P[382]{
   GP1:
	UF : 0, UT : 1,		CONFIG : 'N U T, 0, 0, 0',
	X =	1901.936766	mm,	Y =	727.255833	mm,	Z =	782.023540	mm,
	W =	-151.714705	deg,	P =	-51.403130	deg,	R =	86.436087	deg
};
P[383]{
   GP1:
	UF : 0, UT : 1,		CONFIG : 'N U T, 0, 0, 0',
	X =	1885.131021	mm,	Y =	717.571438	mm,	Z =	785.030103	mm,
	W =	-147.037443	deg,	P =	-51.128385	deg,	R =	85.635377	deg
};
P[384]{
   GP1:
	UF : 0, UT : 1,		CONFIG : 'N U T, 0, 0, 0',
	X =	1869.049725	mm,	Y =	707.056034	mm,	Z =	788.968292	mm,
	W =	-142.293668	deg,	P =	-50.578645	deg,	R =	84.961258	deg
};
P[385]{
   GP1:
	UF : 0, UT : 1,		CONFIG : 'N U T, 0, 0, 0',
	X =	1853.457899	mm,	Y =	695.952416	mm,	Z =	793.610294	mm,
	W =	-139.371378	deg,	P =	-49.801635	deg,	R =	84.946616	deg
};
P[386]{
   GP1:
	UF : 0, UT : 1,		CONFIG : 'N U T, 0, 0, 0',
	X =	1838.594903	mm,	Y =	684.232405	mm,	Z =	798.951702	mm,
	W =	-135.684529	deg,	P =	-49.179213	deg,	R =	84.598217	deg
};
P[387]{
   GP1:
	UF : 0, UT : 1,		CONFIG : 'N U T, 0, 0, 0',
	X =	1824.247050	mm,	Y =	672.047896	mm,	Z =	804.854588	mm,
	W =	-133.003710	deg,	P =	-48.647484	deg,	R =	84.428097	deg
};
P[388]{
   GP1:
	UF : 0, UT : 1,		CONFIG : 'N U T, 0, 0, 0',
	X =	1810.719043	mm,	Y =	659.440410	mm,	Z =	811.371247	mm,
	W =	-129.945774	deg,	P =	-47.843357	deg,	R =	84.483658	deg
};
P[389]{
   GP1:
	UF : 0, UT : 1,		CONFIG : 'N U T, 0, 0, 0',
	X =	1804.034364	mm,	Y =	652.928161	mm,	Z =	814.783583	mm,
	W =	-128.085999	deg,	P =	-47.790016	deg,	R =	83.961023	deg
};
P[390]{
   GP1:
	UF : 0, UT : 1,		CONFIG : 'N U T, 0, 0, 0',
	X =	1805.489552	mm,	Y =	648.057612	mm,	Z =	805.993139	mm,
	W =	-118.280441	deg,	P =	-25.249973	deg,	R =	66.929569	deg
};
P[391]{
   GP1:
	UF : 0, UT : 1,		CONFIG : 'N U T, 0, 0, 0',
	X =	1812.203439	mm,	Y =	654.534929	mm,	Z =	802.566706	mm,
	W =	-118.280441	deg,	P =	-25.249973	deg,	R =	66.929569	deg
};
P[392]{
   GP1:
	UF : 0, UT : 1,		CONFIG : 'N U T, 0, 0, 0',
	X =	1825.953302	mm,	Y =	667.117557	mm,	Z =	796.150605	mm,
	W =	-119.553021	deg,	P =	-25.967899	deg,	R =	66.217655	deg
};
P[393]{
   GP1:
	UF : 0, UT : 1,		CONFIG : 'N U T, 0, 0, 0',
	X =	1840.283003	mm,	Y =	679.245035	mm,	Z =	790.296569	mm,
	W =	-121.343606	deg,	P =	-27.066084	deg,	R =	65.126643	deg
};
P[394]{
   GP1:
	UF : 0, UT : 1,		CONFIG : 'N U T, 0, 0, 0',
	X =	1855.178855	mm,	Y =	690.957511	mm,	Z =	785.030157	mm,
	W =	-123.834308	deg,	P =	-27.839914	deg,	R =	64.621906	deg
};
P[395]{
   GP1:
	UF : 0, UT : 1,		CONFIG : 'N U T, 0, 0, 0',
	X =	1870.722402	mm,	Y =	702.006487	mm,	Z =	780.427067	mm,
	W =	-125.757358	deg,	P =	-29.362690	deg,	R =	63.090015	deg
};
P[396]{
   GP1:
	UF : 0, UT : 1,		CONFIG : 'N U T, 0, 0, 0',
	X =	1886.912120	mm,	Y =	712.361926	mm,	Z =	776.544794	mm,
	W =	-127.137960	deg,	P =	-31.279411	deg,	R =	61.084884	deg
};
P[397]{
   GP1:
	UF : 0, UT : 1,		CONFIG : 'N U T, 0, 0, 0',
	X =	1903.741024	mm,	Y =	721.914625	mm,	Z =	773.719192	mm,
	W =	-130.946538	deg,	P =	-32.608966	deg,	R =	60.232135	deg
};
P[398]{
   GP1:
	UF : 0, UT : 1,		CONFIG : 'N U T, 0, 0, 0',
	X =	1921.157911	mm,	Y =	730.631468	mm,	Z =	771.649972	mm,
	W =	-133.177286	deg,	P =	-34.370572	deg,	R =	58.698336	deg
};
P[399]{
   GP1:
	UF : 0, UT : 1,		CONFIG : 'N U T, 0, 0, 0',
	X =	1939.106460	mm,	Y =	738.185459	mm,	Z =	770.748033	mm,
	W =	-136.382473	deg,	P =	-36.661003	deg,	R =	56.846048	deg
};
P[400]{
   GP1:
	UF : 0, UT : 1,		CONFIG : 'N U T, 0, 0, 0',
	X =	1957.509282	mm,	Y =	744.705160	mm,	Z =	770.921949	mm,
	W =	-140.117439	deg,	P =	-38.294588	deg,	R =	55.735219	deg
};
P[401]{
   GP1:
	UF : 0, UT : 1,		CONFIG : 'N U T, 0, 0, 0',
	X =	1976.233128	mm,	Y =	749.875221	mm,	Z =	772.261698	mm,
	W =	-143.501798	deg,	P =	-40.756036	deg,	R =	53.888603	deg
};
P[402]{
   GP1:
	UF : 0, UT : 1,		CONFIG : 'N U T, 0, 0, 0',
	X =	1995.151040	mm,	Y =	753.608286	mm,	Z =	774.825499	mm,
	W =	-146.537598	deg,	P =	-43.694495	deg,	R =	51.728917	deg
};
P[403]{
   GP1:
	UF : 0, UT : 1,		CONFIG : 'N U T, 0, 0, 0',
	X =	2014.131662	mm,	Y =	756.050102	mm,	Z =	778.522436	mm,
	W =	-149.631146	deg,	P =	-46.183910	deg,	R =	50.037999	deg
};
P[404]{
   GP1:
	UF : 0, UT : 1,		CONFIG : 'N U T, 0, 0, 0',
	X =	2032.817354	mm,	Y =	756.903352	mm,	Z =	783.674625	mm,
	W =	-155.609996	deg,	P =	-47.899495	deg,	R =	49.040964	deg
};
P[405]{
   GP1:
	UF : 0, UT : 1,		CONFIG : 'N U T, 0, 0, 0',
	X =	2051.302092	mm,	Y =	756.193182	mm,	Z =	789.739862	mm,
	W =	-157.425664	deg,	P =	-51.603070	deg,	R =	46.654443	deg
};
P[406]{
   GP1:
	UF : 0, UT : 1,		CONFIG : 'N U T, 0, 0, 0',
	X =	2069.427420	mm,	Y =	754.378399	mm,	Z =	796.789881	mm,
	W =	-160.571018	deg,	P =	-53.566344	deg,	R =	45.491306	deg
};
P[407]{
   GP1:
	UF : 0, UT : 1,		CONFIG : 'N U T, 0, 0, 0',
	X =	2086.942757	mm,	Y =	751.238839	mm,	Z =	804.750806	mm,
	W =	-163.790463	deg,	P =	-56.037649	deg,	R =	44.063831	deg
};
P[408]{
   GP1:
	UF : 0, UT : 1,		CONFIG : 'N U T, 0, 0, 0',
	X =	2103.734538	mm,	Y =	746.847799	mm,	Z =	813.628016	mm,
	W =	-167.805714	deg,	P =	-57.866850	deg,	R =	42.962546	deg
};
P[409]{
   GP1:
	UF : 0, UT : 1,		CONFIG : 'N U T, 0, 0, 0',
	X =	2120.121828	mm,	Y =	741.533562	mm,	Z =	823.012356	mm,
	W =	-169.515653	deg,	P =	-59.824191	deg,	R =	41.934243	deg
};
P[410]{
   GP1:
	UF : 0, UT : 1,		CONFIG : 'N U T, 0, 0, 0',
	X =	2135.809632	mm,	Y =	735.266252	mm,	Z =	832.922306	mm,
	W =	-170.897609	deg,	P =	-62.624007	deg,	R =	40.637323	deg
};
P[411]{
   GP1:
	UF : 0, UT : 1,		CONFIG : 'N U T, 0, 0, 0',
	X =	2150.697320	mm,	Y =	728.173791	mm,	Z =	843.480209	mm,
	W =	-174.130853	deg,	P =	-63.898821	deg,	R =	39.881575	deg
};
P[412]{
   GP1:
	UF : 0, UT : 1,		CONFIG : 'N U T, 0, 0, 0',
	X =	2165.138622	mm,	Y =	720.374642	mm,	Z =	854.327618	mm,
	W =	-175.204728	deg,	P =	-65.758106	deg,	R =	39.148980	deg
};
P[413]{
   GP1:
	UF : 0, UT : 1,		CONFIG : 'N U T, 0, 0, 0',
	X =	2178.740148	mm,	Y =	711.855194	mm,	Z =	865.589791	mm,
	W =	-177.331694	deg,	P =	-67.680964	deg,	R =	38.363196	deg
};
P[414]{
   GP1:
	UF : 0, UT : 1,		CONFIG : 'N U T, 0, 0, 0',
	X =	2191.774572	mm,	Y =	702.742815	mm,	Z =	877.172249	mm,
	W =	-178.961511	deg,	P =	-69.127925	deg,	R =	37.827748	deg
};
P[415]{
   GP1:
	UF : 0, UT : 1,		CONFIG : 'N U T, 0, 0, 0',
	X =	2186.634600	mm,	Y =	701.073329	mm,	Z =	863.753783	mm,
	W =	133.613067	deg,	P =	-56.139818	deg,	R =	90.707230	deg
};
P[416]{
   GP1:
	UF : 0, UT : 1,		CONFIG : 'N U T, 0, 0, 0',
	X =	2173.210709	mm,	Y =	710.002963	mm,	Z =	852.229285	mm,
	W =	133.613067	deg,	P =	-56.139818	deg,	R =	90.707230	deg
};
P[417]{
   GP1:
	UF : 0, UT : 1,		CONFIG : 'N U T, 0, 0, 0',
	X =	2159.155826	mm,	Y =	718.028851	mm,	Z =	841.201692	mm,
	W =	136.846302	deg,	P =	-55.948190	deg,	R =	91.020186	deg
};
P[418]{
   GP1:
	UF : 0, UT : 1,		CONFIG : 'N U T, 0, 0, 0',
	X =	2144.534743	mm,	Y =	725.561610	mm,	Z =	830.433379	mm,
	W =	139.007318	deg,	P =	-55.906508	deg,	R =	91.308868	deg
};
P[419]{
   GP1:
	UF : 0, UT : 1,		CONFIG : 'N U T, 0, 0, 0',
	X =	2129.236263	mm,	Y =	732.215606	mm,	Z =	820.204356	mm,
	W =	142.641369	deg,	P =	-55.588173	deg,	R =	91.285535	deg
};
P[420]{
   GP1:
	UF : 0, UT : 1,		CONFIG : 'N U T, 0, 0, 0',
	X =	2113.285254	mm,	Y =	738.059573	mm,	Z =	810.455841	mm,
	W =	146.014779	deg,	P =	-55.372652	deg,	R =	91.325542	deg
};
P[421]{
   GP1:
	UF : 0, UT : 1,		CONFIG : 'N U T, 0, 0, 0',
	X =	2096.698526	mm,	Y =	742.938558	mm,	Z =	801.332479	mm,
	W =	149.978045	deg,	P =	-55.027116	deg,	R =	91.206586	deg
};
P[422]{
   GP1:
	UF : 0, UT : 1,		CONFIG : 'N U T, 0, 0, 0',
	X =	2079.499669	mm,	Y =	746.762081	mm,	Z =	792.911791	mm,
	W =	154.264576	deg,	P =	-54.635969	deg,	R =	91.033179	deg
};
P[423]{
   GP1:
	UF : 0, UT : 1,		CONFIG : 'N U T, 0, 0, 0',
	X =	2061.718554	mm,	Y =	749.294435	mm,	Z =	785.384968	mm,
	W =	159.358992	deg,	P =	-54.241219	deg,	R =	90.849508	deg
};
P[424]{
   GP1:
	UF : 0, UT : 1,		CONFIG : 'N U T, 0, 0, 0',
	X =	2043.468705	mm,	Y =	750.695013	mm,	Z =	778.604240	mm,
	W =	163.651309	deg,	P =	-54.643114	deg,	R =	91.026912	deg
};
P[425]{
   GP1:
	UF : 0, UT : 1,		CONFIG : 'N U T, 0, 0, 0',
	X =	2024.862362	mm,	Y =	750.526321	mm,	Z =	773.152849	mm,
	W =	170.177142	deg,	P =	-53.461414	deg,	R =	90.339652	deg
};
P[426]{
   GP1:
	UF : 0, UT : 1,		CONFIG : 'N U T, 0, 0, 0',
	X =	2005.984397	mm,	Y =	748.955899	mm,	Z =	768.770108	mm,
	W =	175.722594	deg,	P =	-52.709076	deg,	R =	89.957307	deg
};
P[427]{
   GP1:
	UF : 0, UT : 1,		CONFIG : 'N U T, 0, 0, 0',
	X =	1987.047314	mm,	Y =	746.010534	mm,	Z =	765.364078	mm,
	W =	-178.653351	deg,	P =	-53.676796	deg,	R =	89.597607	deg
};
P[428]{
   GP1:
	UF : 0, UT : 1,		CONFIG : 'N U T, 0, 0, 0',
	X =	1968.269258	mm,	Y =	741.589641	mm,	Z =	763.449879	mm,
	W =	-172.301934	deg,	P =	-52.215645	deg,	R =	89.108243	deg
};
P[429]{
   GP1:
	UF : 0, UT : 1,		CONFIG : 'N U T, 0, 0, 0',
	X =	1949.683228	mm,	Y =	735.867392	mm,	Z =	762.574025	mm,
	W =	-166.727696	deg,	P =	-52.147337	deg,	R =	88.499624	deg
};
P[430]{
   GP1:
	UF : 0, UT : 1,		CONFIG : 'N U T, 0, 0, 0',
	X =	1931.537687	mm,	Y =	728.906759	mm,	Z =	762.984667	mm,
	W =	-161.402140	deg,	P =	-50.785190	deg,	R =	88.352660	deg
};
P[431]{
   GP1:
	UF : 0, UT : 1,		CONFIG : 'N U T, 0, 0, 0',
	X =	1913.894369	mm,	Y =	720.759021	mm,	Z =	764.365662	mm,
	W =	-155.472702	deg,	P =	-51.263880	deg,	R =	87.224493	deg
};
P[432]{
   GP1:
	UF : 0, UT : 1,		CONFIG : 'N U T, 0, 0, 0',
	X =	1896.775808	mm,	Y =	711.703886	mm,	Z =	766.784223	mm,
	W =	-150.833605	deg,	P =	-50.652086	deg,	R =	86.780879	deg
};
P[433]{
   GP1:
	UF : 0, UT : 1,		CONFIG : 'N U T, 0, 0, 0',
	X =	1880.295912	mm,	Y =	701.786455	mm,	Z =	770.150545	mm,
	W =	-146.630492	deg,	P =	-49.748494	deg,	R =	86.649965	deg
};
P[434]{
   GP1:
	UF : 0, UT : 1,		CONFIG : 'N U T, 0, 0, 0',
	X =	1864.365138	mm,	Y =	691.155671	mm,	Z =	774.234987	mm,
	W =	-142.794729	deg,	P =	-49.424405	deg,	R =	86.125445	deg
};
P[435]{
   GP1:
	UF : 0, UT : 1,		CONFIG : 'N U T, 0, 0, 0',
	X =	1849.113413	mm,	Y =	679.894582	mm,	Z =	779.109083	mm,
	W =	-139.403776	deg,	P =	-48.562422	deg,	R =	86.186590	deg
};
P[436]{
   GP1:
	UF : 0, UT : 1,		CONFIG : 'N U T, 0, 0, 0',
	X =	1834.491060	mm,	Y =	668.059164	mm,	Z =	784.620839	mm,
	W =	-136.088896	deg,	P =	-48.063889	deg,	R =	85.921463	deg
};
P[437]{
   GP1:
	UF : 0, UT : 1,		CONFIG : 'N U T, 0, 0, 0',
	X =	1820.513635	mm,	Y =	655.728175	mm,	Z =	790.732302	mm,
	W =	-132.837127	deg,	P =	-47.655336	deg,	R =	85.548407	deg
};
P[438]{
   GP1:
	UF : 0, UT : 1,		CONFIG : 'N U T, 0, 0, 0',
	X =	1807.025014	mm,	Y =	643.027015	mm,	Z =	797.323227	mm,
	W =	-130.462952	deg,	P =	-47.253573	deg,	R =	85.381539	deg
};
P[439]{
   GP1:
	UF : 0, UT : 1,		CONFIG : 'N U T, 0, 0, 0',
	X =	1808.632578	mm,	Y =	637.999708	mm,	Z =	788.721272	mm,
	W =	-119.968116	deg,	P =	-24.932390	deg,	R =	67.755263	deg
};
P[440]{
   GP1:
	UF : 0, UT : 1,		CONFIG : 'N U T, 0, 0, 0',
	X =	1815.310699	mm,	Y =	644.342823	mm,	Z =	785.396809	mm,
	W =	-119.968116	deg,	P =	-24.932390	deg,	R =	67.755263	deg
};
P[441]{
   GP1:
	UF : 0, UT : 1,		CONFIG : 'N U T, 0, 0, 0',
	X =	1828.937900	mm,	Y =	656.757079	mm,	Z =	779.075124	mm,
	W =	-120.933291	deg,	P =	-25.503310	deg,	R =	67.152954	deg
};
P[442]{
   GP1:
	UF : 0, UT : 1,		CONFIG : 'N U T, 0, 0, 0',
	X =	1843.195636	mm,	Y =	668.591056	mm,	Z =	773.448643	mm,
	W =	-123.046463	deg,	P =	-26.806027	deg,	R =	65.806724	deg
};
P[443]{
   GP1:
	UF : 0, UT : 1,		CONFIG : 'N U T, 0, 0, 0',
	X =	1858.023543	mm,	Y =	680.021234	mm,	Z =	768.338080	mm,
	W =	-124.862562	deg,	P =	-27.804666	deg,	R =	64.848593	deg
};
P[444]{
   GP1:
	UF : 0, UT : 1,		CONFIG : 'N U T, 0, 0, 0',
	X =	1873.459502	mm,	Y =	690.849611	mm,	Z =	763.968271	mm,
	W =	-127.624928	deg,	P =	-28.905108	deg,	R =	63.936758	deg
};
P[445]{
   GP1:
	UF : 0, UT : 1,		CONFIG : 'N U T, 0, 0, 0',
	X =	1889.485011	mm,	Y =	701.051034	mm,	Z =	760.200825	mm,
	W =	-129.215229	deg,	P =	-30.446290	deg,	R =	62.373977	deg
};
P[446]{
   GP1:
	UF : 0, UT : 1,		CONFIG : 'N U T, 0, 0, 0',
	X =	1906.116311	mm,	Y =	710.431489	mm,	Z =	757.393894	mm,
	W =	-132.248082	deg,	P =	-32.023439	deg,	R =	61.033740	deg
};
P[447]{
   GP1:
	UF : 0, UT : 1,		CONFIG : 'N U T, 0, 0, 0',
	X =	1923.335471	mm,	Y =	718.930100	mm,	Z =	755.412367	mm,
	W =	-134.227112	deg,	P =	-34.097959	deg,	R =	59.112079	deg
};
P[448]{
   GP1:
	UF : 0, UT : 1,		CONFIG : 'N U T, 0, 0, 0',
	X =	1941.074451	mm,	Y =	726.336330	mm,	Z =	754.576473	mm,
	W =	-137.427428	deg,	P =	-36.272612	deg,	R =	57.336758	deg
};
P[449]{
   GP1:
	UF : 0, UT : 1,		CONFIG : 'N U T, 0, 0, 0',
	X =	1959.258358	mm,	Y =	732.705571	mm,	Z =	754.756467	mm,
	W =	-140.534645	deg,	P =	-38.203158	deg,	R =	55.855613	deg
};
P[450]{
   GP1:
	UF : 0, UT : 1,		CONFIG : 'N U T, 0, 0, 0',
	X =	1977.709684	mm,	Y =	737.832473	mm,	Z =	756.240512	mm,
	W =	-145.990036	deg,	P =	-39.401021	deg,	R =	55.158578	deg
};
P[451]{
   GP1:
	UF : 0, UT : 1,		CONFIG : 'N U T, 0, 0, 0',
	X =	1996.381049	mm,	Y =	741.462266	mm,	Z =	758.804472	mm,
	W =	-148.889992	deg,	P =	-42.355562	deg,	R =	52.899958	deg
};
P[452]{
   GP1:
	UF : 0, UT : 1,		CONFIG : 'N U T, 0, 0, 0',
	X =	2015.092255	mm,	Y =	743.714069	mm,	Z =	762.512016	mm,
	W =	-151.386913	deg,	P =	-45.459649	deg,	R =	50.658130	deg
};
P[453]{
   GP1:
	UF : 0, UT : 1,		CONFIG : 'N U T, 0, 0, 0',
	X =	2033.575537	mm,	Y =	744.530955	mm,	Z =	767.544065	mm,
	W =	-156.105006	deg,	P =	-47.514341	deg,	R =	49.297600	deg
};
P[454]{
   GP1:
	UF : 0, UT : 1,		CONFIG : 'N U T, 0, 0, 0',
	X =	2051.909767	mm,	Y =	744.028237	mm,	Z =	773.401509	mm,
	W =	-157.712965	deg,	P =	-50.709484	deg,	R =	47.226454	deg
};
P[455]{
   GP1:
	UF : 0, UT : 1,		CONFIG : 'N U T, 0, 0, 0',
	X =	2069.734694	mm,	Y =	742.344760	mm,	Z =	780.406294	mm,
	W =	-162.712369	deg,	P =	-51.809564	deg,	R =	46.456856	deg
};
P[456]{
   GP1:
	UF : 0, UT : 1,		CONFIG : 'N U T, 0, 0, 0',
	X =	2087.005748	mm,	Y =	739.271998	mm,	Z =	788.272512	mm,
	W =	-166.243157	deg,	P =	-54.030285	deg,	R =	45.002322	deg
};
P[457]{
   GP1:
	UF : 0, UT : 1,		CONFIG : 'N U T, 0, 0, 0',
	X =	2103.757318	mm,	Y =	735.027800	mm,	Z =	796.829129	mm,
	W =	-168.056359	deg,	P =	-56.892944	deg,	R =	43.414639	deg
};
P[458]{
   GP1:
	UF : 0, UT : 1,		CONFIG : 'N U T, 0, 0, 0',
	X =	2119.977430	mm,	Y =	729.932973	mm,	Z =	806.030766	mm,
	W =	-170.353518	deg,	P =	-58.584566	deg,	R =	42.413878	deg
};
P[459]{
   GP1:
	UF : 0, UT : 1,		CONFIG : 'N U T, 0, 0, 0',
	X =	2135.397002	mm,	Y =	723.770676	mm,	Z =	815.837692	mm,
	W =	-172.583524	deg,	P =	-61.187894	deg,	R =	41.070959	deg
};
P[460]{
   GP1:
	UF : 0, UT : 1,		CONFIG : 'N U T, 0, 0, 0',
	X =	2150.284740	mm,	Y =	716.888007	mm,	Z =	826.147103	mm,
	W =	-174.685768	deg,	P =	-62.551246	deg,	R =	40.281326	deg
};
P[461]{
   GP1:
	UF : 0, UT : 1,		CONFIG : 'N U T, 0, 0, 0',
	X =	2164.573262	mm,	Y =	709.275279	mm,	Z =	836.795716	mm,
	W =	-175.969156	deg,	P =	-64.632942	deg,	R =	39.400791	deg
};
P[462]{
   GP1:
	UF : 0, UT : 1,		CONFIG : 'N U T, 0, 0, 0',
	X =	2177.925079	mm,	Y =	701.249794	mm,	Z =	847.562048	mm,
	W =	-177.630447	deg,	P =	-66.197531	deg,	R =	38.690815	deg
};
P[463]{
   GP1:
	UF : 0, UT : 1,		CONFIG : 'N U T, 0, 0, 0',
	X =	2184.886697	mm,	Y =	696.730596	mm,	Z =	853.380883	mm,
	W =	-178.039191	deg,	P =	-67.748396	deg,	R =	38.248582	deg
};
P[464]{
   GP1:
	UF : 0, UT : 1,		CONFIG : 'N U T, 0, 0, 0',
	X =	2181.841525	mm,	Y =	692.988579	mm,	Z =	842.321213	mm,
	W =	135.564305	deg,	P =	-55.691506	deg,	R =	90.246712	deg
};
P[465]{
   GP1:
	UF : 0, UT : 1,		CONFIG : 'N U T, 0, 0, 0',
	X =	2168.105078	mm,	Y =	701.501885	mm,	Z =	831.052627	mm,
	W =	135.564305	deg,	P =	-55.691506	deg,	R =	90.246712	deg
};
P[466]{
   GP1:
	UF : 0, UT : 1,		CONFIG : 'N U T, 0, 0, 0',
	X =	2153.814736	mm,	Y =	709.163986	mm,	Z =	820.243529	mm,
	W =	138.375103	deg,	P =	-55.684306	deg,	R =	90.822111	deg
};
P[467]{
   GP1:
	UF : 0, UT : 1,		CONFIG : 'N U T, 0, 0, 0',
	X =	2138.911970	mm,	Y =	716.321315	mm,	Z =	809.866842	mm,
	W =	142.009492	deg,	P =	-54.264254	deg,	R =	89.229699	deg
};
P[468]{
   GP1:
	UF : 0, UT : 1,		CONFIG : 'N U T, 0, 0, 0',
	X =	2123.403645	mm,	Y =	722.595473	mm,	Z =	799.908879	mm,
	W =	145.312444	deg,	P =	-53.815509	deg,	R =	89.257980	deg
};
P[469]{
   GP1:
	UF : 0, UT : 1,		CONFIG : 'N U T, 0, 0, 0',
	X =	2107.250912	mm,	Y =	727.950334	mm,	Z =	790.506896	mm,
	W =	148.867175	deg,	P =	-53.503316	deg,	R =	89.468764	deg
};
P[470]{
   GP1:
	UF : 0, UT : 1,		CONFIG : 'N U T, 0, 0, 0',
	X =	2090.470478	mm,	Y =	732.371089	mm,	Z =	781.755813	mm,
	W =	152.827145	deg,	P =	-52.676702	deg,	R =	89.200170	deg
};
P[471]{
   GP1:
	UF : 0, UT : 1,		CONFIG : 'N U T, 0, 0, 0',
	X =	2073.108528	mm,	Y =	735.480186	mm,	Z =	773.759699	mm,
	W =	157.137441	deg,	P =	-53.289463	deg,	R =	90.116868	deg
};
P[472]{
   GP1:
	UF : 0, UT : 1,		CONFIG : 'N U T, 0, 0, 0',
	X =	2055.214096	mm,	Y =	737.578414	mm,	Z =	766.529325	mm,
	W =	161.169691	deg,	P =	-53.382060	deg,	R =	90.356757	deg
};
P[473]{
   GP1:
	UF : 0, UT : 1,		CONFIG : 'N U T, 0, 0, 0',
	X =	2036.896888	mm,	Y =	738.343835	mm,	Z =	760.395742	mm,
	W =	166.601688	deg,	P =	-52.199372	deg,	R =	89.929277	deg
};
P[474]{
   GP1:
	UF : 0, UT : 1,		CONFIG : 'N U T, 0, 0, 0',
	X =	2018.275633	mm,	Y =	737.678830	mm,	Z =	755.238471	mm,
	W =	171.923011	deg,	P =	-52.382412	deg,	R =	90.013689	deg
};
P[475]{
   GP1:
	UF : 0, UT : 1,		CONFIG : 'N U T, 0, 0, 0',
	X =	1999.494459	mm,	Y =	735.558937	mm,	Z =	751.328959	mm,
	W =	177.796470	deg,	P =	-51.702149	deg,	R =	89.778960	deg
};
P[476]{
   GP1:
	UF : 0, UT : 1,		CONFIG : 'N U T, 0, 0, 0',
	X =	1980.730933	mm,	Y =	731.943968	mm,	Z =	748.679772	mm,
	W =	-176.234904	deg,	P =	-50.990351	deg,	R =	89.558234	deg
};
P[477]{
   GP1:
	UF : 0, UT : 1,		CONFIG : 'N U T, 0, 0, 0',
	X =	1962.059550	mm,	Y =	727.089251	mm,	Z =	747.086400	mm,
	W =	-171.163504	deg,	P =	-50.614298	deg,	R =	89.334151	deg
};
P[478]{
   GP1:
	UF : 0, UT : 1,		CONFIG : 'N U T, 0, 0, 0',
	X =	1943.811917	mm,	Y =	720.820393	mm,	Z =	746.742659	mm,
	W =	-164.843819	deg,	P =	-50.667597	deg,	R =	88.790665	deg
};
P[479]{
   GP1:
	UF : 0, UT : 1,		CONFIG : 'N U T, 0, 0, 0',
	X =	1925.896158	mm,	Y =	713.478778	mm,	Z =	747.474732	mm,
	W =	-159.962244	deg,	P =	-50.174209	deg,	R =	88.463752	deg
};
P[480]{
   GP1:
	UF : 0, UT : 1,		CONFIG : 'N U T, 0, 0, 0',
	X =	1908.537864	mm,	Y =	705.085861	mm,	Z =	749.294812	mm,
	W =	-155.229156	deg,	P =	-49.250021	deg,	R =	88.390364	deg
};
P[481]{
   GP1:
	UF : 0, UT : 1,		CONFIG : 'N U T, 0, 0, 0',
	X =	1891.722996	mm,	Y =	695.757420	mm,	Z =	751.975957	mm,
	W =	-150.448327	deg,	P =	-49.273447	deg,	R =	87.694411	deg
};
P[482]{
   GP1:
	UF : 0, UT : 1,		CONFIG : 'N U T, 0, 0, 0',
	X =	1875.511504	mm,	Y =	685.668516	mm,	Z =	755.570823	mm,
	W =	-146.634580	deg,	P =	-48.448142	deg,	R =	87.712135	deg
};
P[483]{
   GP1:
	UF : 0, UT : 1,		CONFIG : 'N U T, 0, 0, 0',
	X =	1859.975552	mm,	Y =	674.831135	mm,	Z =	759.944593	mm,
	W =	-142.505365	deg,	P =	-48.089697	deg,	R =	87.292011	deg
};
P[484]{
   GP1:
	UF : 0, UT : 1,		CONFIG : 'N U T, 0, 0, 0',
	X =	1845.052296	mm,	Y =	663.401217	mm,	Z =	765.037013	mm,
	W =	-139.195876	deg,	P =	-47.514091	deg,	R =	87.203760	deg
};
P[485]{
   GP1:
	UF : 0, UT : 1,		CONFIG : 'N U T, 0, 0, 0',
	X =	1830.679097	mm,	Y =	651.487074	mm,	Z =	770.710133	mm,
	W =	-136.478687	deg,	P =	-46.989176	deg,	R =	87.193937	deg
};
P[486]{
   GP1:
	UF : 0, UT : 1,		CONFIG : 'N U T, 0, 0, 0',
	X =	1816.859825	mm,	Y =	639.096963	mm,	Z =	776.918343	mm,
	W =	-133.539043	deg,	P =	-46.703283	deg,	R =	86.858768	deg
};
P[487]{
   GP1:
	UF : 0, UT : 1,		CONFIG : 'N U T, 0, 0, 0',
	X =	1810.198746	mm,	Y =	632.845491	mm,	Z =	780.152938	mm,
	W =	-131.930628	deg,	P =	-46.421710	deg,	R =	86.813093	deg
};
P[488]{
   GP1:
	UF : 0, UT : 1,		CONFIG : 'N U T, 0, 0, 0',
	X =	1811.905570	mm,	Y =	627.582502	mm,	Z =	771.764730	mm,
	W =	-121.363606	deg,	P =	-24.679915	deg,	R =	68.375183	deg
};
P[489]{
   GP1:
	UF : 0, UT : 1,		CONFIG : 'N U T, 0, 0, 0',
	X =	1818.666143	mm,	Y =	633.911365	mm,	Z =	768.477028	mm,
	W =	-121.363606	deg,	P =	-24.679915	deg,	R =	68.375183	deg
};
P[490]{
   GP1:
	UF : 0, UT : 1,		CONFIG : 'N U T, 0, 0, 0',
	X =	1832.401064	mm,	Y =	646.179658	mm,	Z =	762.342043	mm,
	W =	-122.780141	deg,	P =	-25.197941	deg,	R =	67.900015	deg
};
P[491]{
   GP1:
	UF : 0, UT : 1,		CONFIG : 'N U T, 0, 0, 0',
	X =	1846.699673	mm,	Y =	658.005791	mm,	Z =	756.721178	mm,
	W =	-124.437038	deg,	P =	-26.258499	deg,	R =	66.751578	deg
};
P[492]{
   GP1:
	UF : 0, UT : 1,		CONFIG : 'N U T, 0, 0, 0',
	X =	1861.641008	mm,	Y =	669.246542	mm,	Z =	751.765506	mm,
	W =	-126.224273	deg,	P =	-27.726784	deg,	R =	65.160017	deg
};
P[493]{
   GP1:
	UF : 0, UT : 1,		CONFIG : 'N U T, 0, 0, 0',
	X =	1877.185163	mm,	Y =	679.963409	mm,	Z =	747.541220	mm,
	W =	-129.109028	deg,	P =	-28.633967	deg,	R =	64.449103	deg
};
P[494]{
   GP1:
	UF : 0, UT : 1,		CONFIG : 'N U T, 0, 0, 0',
	X =	1893.336367	mm,	Y =	689.966226	mm,	Z =	744.003393	mm,
	W =	-131.145059	deg,	P =	-30.184059	deg,	R =	62.911972	deg
};
P[495]{
   GP1:
	UF : 0, UT : 1,		CONFIG : 'N U T, 0, 0, 0',
	X =	1910.073926	mm,	Y =	699.189762	mm,	Z =	741.308186	mm,
	W =	-133.479291	deg,	P =	-31.880690	deg,	R =	61.321917	deg
};
P[496]{
   GP1:
	UF : 0, UT : 1,		CONFIG : 'N U T, 0, 0, 0',
	X =	1927.359789	mm,	Y =	707.532839	mm,	Z =	739.589631	mm,
	W =	-136.768422	deg,	P =	-33.381058	deg,	R =	60.082388	deg
};
P[497]{
   GP1:
	UF : 0, UT : 1,		CONFIG : 'N U T, 0, 0, 0',
	X =	1945.169599	mm,	Y =	714.763464	mm,	Z =	738.868356	mm,
	W =	-139.296913	deg,	P =	-35.742072	deg,	R =	58.004742	deg
};
P[498]{
   GP1:
	UF : 0, UT : 1,		CONFIG : 'N U T, 0, 0, 0',
	X =	1963.386131	mm,	Y =	720.915378	mm,	Z =	739.257957	mm,
	W =	-142.704252	deg,	P =	-37.648572	deg,	R =	56.501128	deg
};
P[499]{
   GP1:
	UF : 0, UT : 1,		CONFIG : 'N U T, 0, 0, 0',
	X =	1981.873264	mm,	Y =	725.701440	mm,	Z =	740.932512	mm,
	W =	-147.124087	deg,	P =	-39.663573	deg,	R =	54.975846	deg
};
P[500]{
   GP1:
	UF : 0, UT : 1,		CONFIG : 'N U T, 0, 0, 0',
	X =	2000.568180	mm,	Y =	729.249511	mm,	Z =	743.646903	mm,
	W =	-150.477601	deg,	P =	-41.719304	deg,	R =	53.411569	deg
};
P[501]{
   GP1:
	UF : 0, UT : 1,		CONFIG : 'N U T, 0, 0, 0',
	X =	2019.172974	mm,	Y =	731.257679	mm,	Z =	747.673623	mm,
	W =	-154.834890	deg,	P =	-44.104677	deg,	R =	51.631088	deg
};
P[502]{
   GP1:
	UF : 0, UT : 1,		CONFIG : 'N U T, 0, 0, 0',
	X =	2037.736879	mm,	Y =	731.942008	mm,	Z =	752.625278	mm,
	W =	-156.781352	deg,	P =	-47.161624	deg,	R =	49.521897	deg
};
P[503]{
   GP1:
	UF : 0, UT : 1,		CONFIG : 'N U T, 0, 0, 0',
	X =	2055.914550	mm,	Y =	731.278195	mm,	Z =	758.722915	mm,
	W =	-160.313910	deg,	P =	-49.612374	deg,	R =	47.864900	deg
};
P[504]{
   GP1:
	UF : 0, UT : 1,		CONFIG : 'N U T, 0, 0, 0',
	X =	2073.553402	mm,	Y =	729.106124	mm,	Z =	765.891541	mm,
	W =	-163.655904	deg,	P =	-52.580426	deg,	R =	45.969155	deg
};
P[505]{
   GP1:
	UF : 0, UT : 1,		CONFIG : 'N U T, 0, 0, 0',
	X =	2090.853690	mm,	Y =	725.951311	mm,	Z =	773.830626	mm,
	W =	-166.519836	deg,	P =	-54.087477	deg,	R =	44.948519	deg
};
P[506]{
   GP1:
	UF : 0, UT : 1,		CONFIG : 'N U T, 0, 0, 0',
	X =	2107.610690	mm,	Y =	721.817339	mm,	Z =	782.457272	mm,
	W =	-169.611659	deg,	P =	-55.396209	deg,	R =	43.959850	deg
};
P[507]{
   GP1:
	UF : 0, UT : 1,		CONFIG : 'N U T, 0, 0, 0',
	X =	2123.472696	mm,	Y =	716.383569	mm,	Z =	791.830177	mm,
	W =	-172.572596	deg,	P =	-58.108517	deg,	R =	42.321565	deg
};
P[508]{
   GP1:
	UF : 0, UT : 1,		CONFIG : 'N U T, 0, 0, 0',
	X =	2138.990100	mm,	Y =	710.202932	mm,	Z =	801.651689	mm,
	W =	-173.731197	deg,	P =	-59.986051	deg,	R =	41.378752	deg
};
P[509]{
   GP1:
	UF : 0, UT : 1,		CONFIG : 'N U T, 0, 0, 0',
	X =	2153.752955	mm,	Y =	703.175636	mm,	Z =	811.935509	mm,
	W =	-175.164563	deg,	P =	-62.594805	deg,	R =	40.192030	deg
};
P[510]{
   GP1:
	UF : 0, UT : 1,		CONFIG : 'N U T, 0, 0, 0',
	X =	2167.934444	mm,	Y =	695.527109	mm,	Z =	822.646034	mm,
	W =	-176.891181	deg,	P =	-64.081073	deg,	R =	39.413915	deg
};
P[511]{
   GP1:
	UF : 0, UT : 1,		CONFIG : 'N U T, 0, 0, 0',
	X =	2181.580363	mm,	Y =	687.256026	mm,	Z =	833.690767	mm,
	W =	-178.302682	deg,	P =	-65.664938	deg,	R =	38.701290	deg
};
P[512]{
   GP1:
	UF : 0, UT : 1,		CONFIG : 'N U T, 0, 0, 0',
	X =	2181.138489	mm,	Y =	681.541073	mm,	Z =	825.024241	mm,
	W =	137.165595	deg,	P =	-54.783551	deg,	R =	88.900287	deg
};
P[513]{
   GP1:
	UF : 0, UT : 1,		CONFIG : 'N U T, 0, 0, 0',
	X =	2167.219744	mm,	Y =	689.889300	mm,	Z =	813.839668	mm,
	W =	137.165595	deg,	P =	-54.783551	deg,	R =	88.900287	deg
};
P[514]{
   GP1:
	UF : 0, UT : 1,		CONFIG : 'N U T, 0, 0, 0',
	X =	2152.891570	mm,	Y =	697.596031	mm,	Z =	802.996135	mm,
	W =	139.158797	deg,	P =	-54.818348	deg,	R =	89.482178	deg
};
P[515]{
   GP1:
	UF : 0, UT : 1,		CONFIG : 'N U T, 0, 0, 0',
	X =	2137.853717	mm,	Y =	704.535181	mm,	Z =	792.762446	mm,
	W =	143.586391	deg,	P =	-53.130097	deg,	R =	87.951002	deg
};
P[516]{
   GP1:
	UF : 0, UT : 1,		CONFIG : 'N U T, 0, 0, 0',
	X =	2122.222818	mm,	Y =	710.673714	mm,	Z =	782.837928	mm,
	W =	146.229641	deg,	P =	-53.103934	deg,	R =	88.536477	deg
};
P[517]{
   GP1:
	UF : 0, UT : 1,		CONFIG : 'N U T, 0, 0, 0',
	X =	2105.935847	mm,	Y =	715.941000	mm,	Z =	773.609951	mm,
	W =	150.457726	deg,	P =	-51.462751	deg,	R =	87.617398	deg
};
P[518]{
   GP1:
	UF : 0, UT : 1,		CONFIG : 'N U T, 0, 0, 0',
	X =	2089.033459	mm,	Y =	720.029410	mm,	Z =	764.961570	mm,
	W =	154.098297	deg,	P =	-51.794541	deg,	R =	88.616848	deg
};
P[519]{
   GP1:
	UF : 0, UT : 1,		CONFIG : 'N U T, 0, 0, 0',
	X =	2071.566502	mm,	Y =	723.179087	mm,	Z =	757.028896	mm,
	W =	157.832303	deg,	P =	-51.347296	deg,	R =	88.813963	deg
};
P[520]{
   GP1:
	UF : 0, UT : 1,		CONFIG : 'N U T, 0, 0, 0',
	X =	2053.617650	mm,	Y =	724.988818	mm,	Z =	749.983011	mm,
	W =	162.466080	deg,	P =	-51.611491	deg,	R =	89.452096	deg
};
P[521]{
   GP1:
	UF : 0, UT : 1,		CONFIG : 'N U T, 0, 0, 0',
	X =	2035.220444	mm,	Y =	725.408083	mm,	Z =	744.090003	mm,
	W =	167.925319	deg,	P =	-50.586646	deg,	R =	89.402669	deg
};
P[522]{
   GP1:
	UF : 0, UT : 1,		CONFIG : 'N U T, 0, 0, 0',
	X =	2016.523743	mm,	Y =	724.533768	mm,	Z =	739.063885	mm,
	W =	172.613009	deg,	P =	-51.094560	deg,	R =	89.732425	deg
};
P[523]{
   GP1:
	UF : 0, UT : 1,		CONFIG : 'N U T, 0, 0, 0',
	X =	1997.699306	mm,	Y =	722.307135	mm,	Z =	735.322337	mm,
	W =	177.965716	deg,	P =	-49.495082	deg,	R =	89.649080	deg
};
P[524]{
   GP1:
	UF : 0, UT : 1,		CONFIG : 'N U T, 0, 0, 0',
	X =	1978.930103	mm,	Y =	718.562419	mm,	Z =	732.795071	mm,
	W =	-176.418280	deg,	P =	-48.643646	deg,	R =	89.783058	deg
};
P[525]{
   GP1:
	UF : 0, UT : 1,		CONFIG : 'N U T, 0, 0, 0',
	X =	1960.359994	mm,	Y =	713.375202	mm,	Z =	731.329587	mm,
	W =	-170.319625	deg,	P =	-50.045004	deg,	R =	89.413358	deg
};
P[526]{
   GP1:
	UF : 0, UT : 1,		CONFIG : 'N U T, 0, 0, 0',
	X =	1942.130045	mm,	Y =	706.948292	mm,	Z =	731.181869	mm,
	W =	-164.655681	deg,	P =	-49.584028	deg,	R =	89.179519	deg
};
P[527]{
   GP1:
	UF : 0, UT : 1,		CONFIG : 'N U T, 0, 0, 0',
	X =	1924.264017	mm,	Y =	699.451955	mm,	Z =	732.051898	mm,
	W =	-159.916856	deg,	P =	-49.203087	deg,	R =	88.936259	deg
};
P[528]{
   GP1:
	UF : 0, UT : 1,		CONFIG : 'N U T, 0, 0, 0',
	X =	1906.996207	mm,	Y =	690.890327	mm,	Z =	734.017218	mm,
	W =	-155.007980	deg,	P =	-48.510032	deg,	R =	88.817117	deg
};
P[529]{
   GP1:
	UF : 0, UT : 1,		CONFIG : 'N U T, 0, 0, 0',
	X =	1890.274716	mm,	Y =	681.457701	mm,	Z =	736.950281	mm,
	W =	-151.334369	deg,	P =	-47.293390	deg,	R =	89.235312	deg
};
P[530]{
   GP1:
	UF : 0, UT : 1,		CONFIG : 'N U T, 0, 0, 0',
	X =	1874.235773	mm,	Y =	671.136516	mm,	Z =	740.663412	mm,
	W =	-146.406581	deg,	P =	-47.633843	deg,	R =	88.352009	deg
};
P[531]{
   GP1:
	UF : 0, UT : 1,		CONFIG : 'N U T, 0, 0, 0',
	X =	1858.704485	mm,	Y =	660.241574	mm,	Z =	745.137970	mm,
	W =	-143.363223	deg,	P =	-47.025042	deg,	R =	88.426086	deg
};
P[532]{
   GP1:
	UF : 0, UT : 1,		CONFIG : 'N U T, 0, 0, 0',
	X =	1843.833537	mm,	Y =	648.750559	mm,	Z =	750.283485	mm,
	W =	-139.965621	deg,	P =	-46.604545	deg,	R =	88.276486	deg
};
P[533]{
   GP1:
	UF : 0, UT : 1,		CONFIG : 'N U T, 0, 0, 0',
	X =	1829.491772	mm,	Y =	636.788016	mm,	Z =	755.989653	mm,
	W =	-137.194008	deg,	P =	-46.267107	deg,	R =	88.133231	deg
};
P[534]{
   GP1:
	UF : 0, UT : 1,		CONFIG : 'N U T, 0, 0, 0',
	X =	1815.866369	mm,	Y =	624.347869	mm,	Z =	762.302099	mm,
	W =	-133.943972	deg,	P =	-45.876757	deg,	R =	87.935232	deg
};
P[535]{
   GP1:
	UF : 0, UT : 1,		CONFIG : 'N U T, 0, 0, 0',
	X =	1821.339978	mm,	Y =	622.399546	mm,	Z =	752.320456	mm,
	W =	-124.257652	deg,	P =	-24.843060	deg,	R =	68.592784	deg
};
P[536]{
   GP1:
	UF : 0, UT : 1,		CONFIG : 'N U T, 0, 0, 0',
	X =	1835.390935	mm,	Y =	634.758530	mm,	Z =	746.154728	mm,
	W =	-124.257652	deg,	P =	-24.843060	deg,	R =	68.592784	deg
};
P[537]{
   GP1:
	UF : 0, UT : 1,		CONFIG : 'N U T, 0, 0, 0',
	X =	1849.909298	mm,	Y =	646.553730	mm,	Z =	740.605246	mm,
	W =	-125.783143	deg,	P =	-26.039341	deg,	R =	67.220883	deg
};
P[538]{
   GP1:
	UF : 0, UT : 1,		CONFIG : 'N U T, 0, 0, 0',
	X =	1865.009843	mm,	Y =	657.873540	mm,	Z =	735.692168	mm,
	W =	-128.009528	deg,	P =	-27.017846	deg,	R =	66.257580	deg
};
P[539]{
   GP1:
	UF : 0, UT : 1,		CONFIG : 'N U T, 0, 0, 0',
	X =	1880.742374	mm,	Y =	668.522121	mm,	Z =	731.433330	mm,
	W =	-129.457693	deg,	P =	-28.742330	deg,	R =	64.362873	deg
};
P[540]{
   GP1:
	UF : 0, UT : 1,		CONFIG : 'N U T, 0, 0, 0',
	X =	1897.098970	mm,	Y =	678.482212	mm,	Z =	728.162659	mm,
	W =	-133.490324	deg,	P =	-29.567881	deg,	R =	63.800246	deg
};
P[541]{
   GP1:
	UF : 0, UT : 1,		CONFIG : 'N U T, 0, 0, 0',
	X =	1914.051490	mm,	Y =	687.668142	mm,	Z =	725.598218	mm,
	W =	-136.063153	deg,	P =	-30.904135	deg,	R =	62.540269	deg
};
P[542]{
   GP1:
	UF : 0, UT : 1,		CONFIG : 'N U T, 0, 0, 0',
	X =	1931.577178	mm,	Y =	695.769845	mm,	Z =	724.073160	mm,
	W =	-138.779969	deg,	P =	-33.104672	deg,	R =	60.478098	deg
};
P[543]{
   GP1:
	UF : 0, UT : 1,		CONFIG : 'N U T, 0, 0, 0',
	X =	1949.594277	mm,	Y =	702.954782	mm,	Z =	723.508579	mm,
	W =	-141.633390	deg,	P =	-34.814724	deg,	R =	58.985453	deg
};
P[544]{
   GP1:
	UF : 0, UT : 1,		CONFIG : 'N U T, 0, 0, 0',
	X =	1967.975807	mm,	Y =	708.813190	mm,	Z =	724.246717	mm,
	W =	-145.986930	deg,	P =	-36.743970	deg,	R =	57.367342	deg
};
P[545]{
   GP1:
	UF : 0, UT : 1,		CONFIG : 'N U T, 0, 0, 0',
	X =	1986.690994	mm,	Y =	713.485803	mm,	Z =	725.976885	mm,
	W =	-148.792688	deg,	P =	-38.954600	deg,	R =	55.553351	deg
};
P[546]{
   GP1:
	UF : 0, UT : 1,		CONFIG : 'N U T, 0, 0, 0',
	X =	2005.460715	mm,	Y =	716.709881	mm,	Z =	729.042109	mm,
	W =	-153.162353	deg,	P =	-41.082741	deg,	R =	53.832137	deg
};
P[547]{
   GP1:
	UF : 0, UT : 1,		CONFIG : 'N U T, 0, 0, 0',
	X =	2024.262891	mm,	Y =	718.600235	mm,	Z =	733.173859	mm,
	W =	-156.478471	deg,	P =	-43.300004	deg,	R =	52.109259	deg
};
P[548]{
   GP1:
	UF : 0, UT : 1,		CONFIG : 'N U T, 0, 0, 0',
	X =	2042.780225	mm,	Y =	718.838354	mm,	Z =	738.506908	mm,
	W =	-159.254519	deg,	P =	-46.915692	deg,	R =	49.584607	deg
};
P[549]{
   GP1:
	UF : 0, UT : 1,		CONFIG : 'N U T, 0, 0, 0',
	X =	2060.996090	mm,	Y =	717.786583	mm,	Z =	744.922635	mm,
	W =	-162.416350	deg,	P =	-49.334115	deg,	R =	47.903588	deg
};
P[550]{
   GP1:
	UF : 0, UT : 1,		CONFIG : 'N U T, 0, 0, 0',
	X =	2078.798334	mm,	Y =	715.534828	mm,	Z =	752.231905	mm,
	W =	-165.403747	deg,	P =	-51.416481	deg,	R =	46.464422	deg
};
P[551]{
   GP1:
	UF : 0, UT : 1,		CONFIG : 'N U T, 0, 0, 0',
	X =	2095.955906	mm,	Y =	712.031539	mm,	Z =	760.456728	mm,
	W =	-169.055675	deg,	P =	-53.276681	deg,	R =	45.051963	deg
};
P[552]{
   GP1:
	UF : 0, UT : 1,		CONFIG : 'N U T, 0, 0, 0',
	X =	2112.642546	mm,	Y =	707.476231	mm,	Z =	769.310594	mm,
	W =	-171.117458	deg,	P =	-55.409733	deg,	R =	43.728895	deg
};
P[553]{
   GP1:
	UF : 0, UT : 1,		CONFIG : 'N U T, 0, 0, 0',
	X =	2128.714028	mm,	Y =	702.010319	mm,	Z =	778.789707	mm,
	W =	-173.494305	deg,	P =	-57.119217	deg,	R =	42.562970	deg
};
P[554]{
   GP1:
	UF : 0, UT : 1,		CONFIG : 'N U T, 0, 0, 0',
	X =	2143.992072	mm,	Y =	695.451866	mm,	Z =	788.801150	mm,
	W =	-174.899258	deg,	P =	-60.366912	deg,	R =	41.029481	deg
};
P[555]{
   GP1:
	UF : 0, UT : 1,		CONFIG : 'N U T, 0, 0, 0',
	X =	2158.843125	mm,	Y =	688.280890	mm,	Z =	799.248934	mm,
	W =	-175.941914	deg,	P =	-62.183292	deg,	R =	40.194389	deg
};
P[556]{
   GP1:
	UF : 0, UT : 1,		CONFIG : 'N U T, 0, 0, 0',
	X =	2172.485016	mm,	Y =	680.677442	mm,	Z =	809.818048	mm,
	W =	-178.309239	deg,	P =	-63.480861	deg,	R =	39.283257	deg
};
P[557]{
   GP1:
	UF : 0, UT : 1,		CONFIG : 'N U T, 0, 0, 0',
	X =	2179.771323	mm,	Y =	676.276925	mm,	Z =	815.698039	mm,
	W =	-179.168365	deg,	P =	-64.558946	deg,	R =	38.781140	deg
};
P[558]{
   GP1:
	UF : 0, UT : 1,		CONFIG : 'N U T, 0, 0, 0',
	X =	2172.448483	mm,	Y =	674.526549	mm,	Z =	801.643526	mm,
	W =	139.757218	deg,	P =	-53.369479	deg,	R =	87.176905	deg
};
P[559]{
   GP1:
	UF : 0, UT : 1,		CONFIG : 'N U T, 0, 0, 0',
	X =	2164.801470	mm,	Y =	678.807783	mm,	Z =	795.755079	mm,
	W =	139.757218	deg,	P =	-53.369479	deg,	R =	87.176905	deg
};
P[560]{
   GP1:
	UF : 0, UT : 1,		CONFIG : 'N U T, 0, 0, 0',
	X =	2150.523545	mm,	Y =	686.109517	mm,	Z =	785.337507	mm,
	W =	141.779192	deg,	P =	-52.892982	deg,	R =	87.075567	deg
};
P[561]{
   GP1:
	UF : 0, UT : 1,		CONFIG : 'N U T, 0, 0, 0',
	X =	2135.245274	mm,	Y =	692.932587	mm,	Z =	774.982974	mm,
	W =	144.397280	deg,	P =	-52.537085	deg,	R =	87.350034	deg
};
P[562]{
   GP1:
	UF : 0, UT : 1,		CONFIG : 'N U T, 0, 0, 0',
	X =	2119.278313	mm,	Y =	698.820062	mm,	Z =	765.230469	mm,
	W =	148.114893	deg,	P =	-51.752348	deg,	R =	87.367444	deg
};
P[563]{
   GP1:
	UF : 0, UT : 1,		CONFIG : 'N U T, 0, 0, 0',
	X =	2102.686383	mm,	Y =	703.845237	mm,	Z =	756.018877	mm,
	W =	151.495508	deg,	P =	-51.017093	deg,	R =	87.416536	deg
};
P[564]{
   GP1:
	UF : 0, UT : 1,		CONFIG : 'N U T, 0, 0, 0',
	X =	2085.512795	mm,	Y =	707.804734	mm,	Z =	747.434083	mm,
	W =	155.012838	deg,	P =	-51.062985	deg,	R =	88.170152	deg
};
P[565]{
   GP1:
	UF : 0, UT : 1,		CONFIG : 'N U T, 0, 0, 0',
	X =	2067.734353	mm,	Y =	710.545304	mm,	Z =	739.810771	mm,
	W =	159.778129	deg,	P =	-49.780882	deg,	R =	88.097988	deg
};
P[566]{
   GP1:
	UF : 0, UT : 1,		CONFIG : 'N U T, 0, 0, 0',
	X =	2049.478100	mm,	Y =	712.044144	mm,	Z =	732.942884	mm,
	W =	163.878111	deg,	P =	-50.046807	deg,	R =	88.820681	deg
};
P[567]{
   GP1:
	UF : 0, UT : 1,		CONFIG : 'N U T, 0, 0, 0',
	X =	2030.834453	mm,	Y =	712.061084	mm,	Z =	727.332459	mm,
	W =	169.426200	deg,	P =	-48.733326	deg,	R =	88.960733	deg
};
P[568]{
   GP1:
	UF : 0, UT : 1,		CONFIG : 'N U T, 0, 0, 0',
	X =	2011.914047	mm,	Y =	710.738243	mm,	Z =	722.681289	mm,
	W =	174.123061	deg,	P =	-48.502819	deg,	R =	89.351106	deg
};
P[569]{
   GP1:
	UF : 0, UT : 1,		CONFIG : 'N U T, 0, 0, 0',
	X =	1992.967315	mm,	Y =	707.860461	mm,	Z =	719.258775	mm,
	W =	179.900303	deg,	P =	-48.816687	deg,	R =	89.690444	deg
};
P[570]{
   GP1:
	UF : 0, UT : 1,		CONFIG : 'N U T, 0, 0, 0',
	X =	1974.020138	mm,	Y =	703.741578	mm,	Z =	717.028742	mm,
	W =	-175.305359	deg,	P =	-47.746908	deg,	R =	89.910278	deg
};
P[571]{
   GP1:
	UF : 0, UT : 1,		CONFIG : 'N U T, 0, 0, 0',
	X =	1955.427942	mm,	Y =	698.071747	mm,	Z =	716.038071	mm,
	W =	-169.073900	deg,	P =	-48.245697	deg,	R =	89.835786	deg
};
P[572]{
   GP1:
	UF : 0, UT : 1,		CONFIG : 'N U T, 0, 0, 0',
	X =	1937.102614	mm,	Y =	691.297711	mm,	Z =	716.219092	mm,
	W =	-164.534112	deg,	P =	-47.297055	deg,	R =	90.059825	deg
};
P[573]{
   GP1:
	UF : 0, UT : 1,		CONFIG : 'N U T, 0, 0, 0',
	X =	1919.373288	mm,	Y =	683.255360	mm,	Z =	717.507870	mm,
	W =	-158.792038	deg,	P =	-47.589528	deg,	R =	89.674772	deg
};
P[574]{
   GP1:
	UF : 0, UT : 1,		CONFIG : 'N U T, 0, 0, 0',
	X =	1902.120784	mm,	Y =	674.289308	mm,	Z =	719.801763	mm,
	W =	-154.437262	deg,	P =	-47.219022	deg,	R =	89.574353	deg
};
P[575]{
   GP1:
	UF : 0, UT : 1,		CONFIG : 'N U T, 0, 0, 0',
	X =	1885.482455	mm,	Y =	664.465084	mm,	Z =	723.027009	mm,
	W =	-150.395360	deg,	P =	-46.611223	deg,	R =	89.641447	deg
};
P[576]{
   GP1:
	UF : 0, UT : 1,		CONFIG : 'N U T, 0, 0, 0',
	X =	1869.470130	mm,	Y =	653.871948	mm,	Z =	727.051099	mm,
	W =	-146.429711	deg,	P =	-46.383313	deg,	R =	89.409407	deg
};
P[577]{
   GP1:
	UF : 0, UT : 1,		CONFIG : 'N U T, 0, 0, 0',
	X =	1854.003475	mm,	Y =	642.694090	mm,	Z =	731.786078	mm,
	W =	-143.497932	deg,	P =	-45.791206	deg,	R =	89.588858	deg
};
P[578]{
   GP1:
	UF : 0, UT : 1,		CONFIG : 'N U T, 0, 0, 0',
	X =	1839.290905	mm,	Y =	630.901908	mm,	Z =	737.248693	mm,
	W =	-140.081460	deg,	P =	-45.220618	deg,	R =	89.713685	deg
};
P[579]{
   GP1:
	UF : 0, UT : 1,		CONFIG : 'N U T, 0, 0, 0',
	X =	1825.112873	mm,	Y =	618.611600	mm,	Z =	743.239229	mm,
	W =	-136.993181	deg,	P =	-45.237351	deg,	R =	89.240232	deg
};
P[580]{
   GP1:
	UF : 0, UT : 1,		CONFIG : 'N U T, 0, 0, 0',
	X =	1824.231261	mm,	Y =	610.542823	mm,	Z =	736.440188	mm,
	W =	-124.873525	deg,	P =	-24.173949	deg,	R =	69.565832	deg
};
P[581]{
   GP1:
	UF : 0, UT : 1,		CONFIG : 'N U T, 0, 0, 0',
	X =	1831.134355	mm,	Y =	616.711356	mm,	Z =	733.329868	mm,
	W =	-124.873525	deg,	P =	-24.173949	deg,	R =	69.565832	deg
};
P[582]{
   GP1:
	UF : 0, UT : 1,		CONFIG : 'N U T, 0, 0, 0',
	X =	1845.348889	mm,	Y =	628.626176	mm,	Z =	727.635363	mm,
	W =	-126.621354	deg,	P =	-24.916556	deg,	R =	68.759910	deg
};
P[583]{
   GP1:
	UF : 0, UT : 1,		CONFIG : 'N U T, 0, 0, 0',
	X =	1860.145551	mm,	Y =	640.004656	mm,	Z =	722.559496	mm,
	W =	-128.681569	deg,	P =	-26.005899	deg,	R =	67.563156	deg
};
P[584]{
   GP1:
	UF : 0, UT : 1,		CONFIG : 'N U T, 0, 0, 0',
	X =	1875.504137	mm,	Y =	650.900841	mm,	Z =	718.112069	mm,
	W =	-131.226089	deg,	P =	-26.775914	deg,	R =	66.812471	deg
};
P[585]{
   GP1:
	UF : 0, UT : 1,		CONFIG : 'N U T, 0, 0, 0',
	X =	1891.482681	mm,	Y =	661.069298	mm,	Z =	714.395745	mm,
	W =	-133.478709	deg,	P =	-28.235203	deg,	R =	65.265321	deg
};
P[586]{
   GP1:
	UF : 0, UT : 1,		CONFIG : 'N U T, 0, 0, 0',
	X =	1908.047786	mm,	Y =	670.518770	mm,	Z =	711.457222	mm,
	W =	-135.707371	deg,	P =	-29.758919	deg,	R =	63.717538	deg
};
P[587]{
   GP1:
	UF : 0, UT : 1,		CONFIG : 'N U T, 0, 0, 0',
	X =	1925.206276	mm,	Y =	678.997374	mm,	Z =	709.433190	mm,
	W =	-137.496161	deg,	P =	-32.164830	deg,	R =	61.337119	deg
};
P[588]{
   GP1:
	UF : 0, UT : 1,		CONFIG : 'N U T, 0, 0, 0',
	X =	1942.863402	mm,	Y =	686.556513	mm,	Z =	708.552673	mm,
	W =	-141.648651	deg,	P =	-33.367195	deg,	R =	60.316431	deg
};
P[589]{
   GP1:
	UF : 0, UT : 1,		CONFIG : 'N U T, 0, 0, 0',
	X =	1960.978697	mm,	Y =	692.978970	mm,	Z =	708.652172	mm,
	W =	-144.681894	deg,	P =	-35.357918	deg,	R =	58.551426	deg
};
P[590]{
   GP1:
	UF : 0, UT : 1,		CONFIG : 'N U T, 0, 0, 0',
	X =	1979.380893	mm,	Y =	698.204726	mm,	Z =	710.016418	mm,
	W =	-149.716121	deg,	P =	-36.468959	deg,	R =	57.499082	deg
};
P[591]{
   GP1:
	UF : 0, UT : 1,		CONFIG : 'N U T, 0, 0, 0',
	X =	1998.019637	mm,	Y =	702.047679	mm,	Z =	712.423469	mm,
	W =	-152.784194	deg,	P =	-38.911678	deg,	R =	55.447053	deg
};
P[592]{
   GP1:
	UF : 0, UT : 1,		CONFIG : 'N U T, 0, 0, 0',
	X =	2016.667589	mm,	Y =	704.354762	mm,	Z =	716.048551	mm,
	W =	-155.393063	deg,	P =	-42.333005	deg,	R =	52.835617	deg
};
P[593]{
   GP1:
	UF : 0, UT : 1,		CONFIG : 'N U T, 0, 0, 0',
	X =	2035.168306	mm,	Y =	705.325302	mm,	Z =	720.930588	mm,
	W =	-159.560545	deg,	P =	-44.296664	deg,	R =	51.218672	deg
};
P[594]{
   GP1:
	UF : 0, UT : 1,		CONFIG : 'N U T, 0, 0, 0',
	X =	2053.502816	mm,	Y =	705.033488	mm,	Z =	726.696422	mm,
	W =	-162.018352	deg,	P =	-46.759808	deg,	R =	49.458695	deg
};
P[595]{
   GP1:
	UF : 0, UT : 1,		CONFIG : 'N U T, 0, 0, 0',
	X =	2071.344304	mm,	Y =	703.424961	mm,	Z =	733.543619	mm,
	W =	-165.926992	deg,	P =	-48.677900	deg,	R =	47.882397	deg
};
P[596]{
   GP1:
	UF : 0, UT : 1,		CONFIG : 'N U T, 0, 0, 0',
	X =	2088.682150	mm,	Y =	700.468799	mm,	Z =	741.237613	mm,
	W =	-168.397673	deg,	P =	-51.508182	deg,	R =	46.027283	deg
};
P[597]{
   GP1:
	UF : 0, UT : 1,		CONFIG : 'N U T, 0, 0, 0',
	X =	2105.415038	mm,	Y =	696.408191	mm,	Z =	749.799292	mm,
	W =	-171.729773	deg,	P =	-53.164498	deg,	R =	44.630312	deg
};
P[598]{
   GP1:
	UF : 0, UT : 1,		CONFIG : 'N U T, 0, 0, 0',
	X =	2121.782519	mm,	Y =	691.548869	mm,	Z =	758.874629	mm,
	W =	-173.853140	deg,	P =	-54.276831	deg,	R =	43.665261	deg
};
P[599]{
   GP1:
	UF : 0, UT : 1,		CONFIG : 'N U T, 0, 0, 0',
	X =	2137.330657	mm,	Y =	685.493206	mm,	Z =	768.463065	mm,
	W =	-174.648553	deg,	P =	-58.314243	deg,	R =	41.851314	deg
};
P[600]{
   GP1:
	UF : 0, UT : 1,		CONFIG : 'N U T, 0, 0, 0',
	X =	2152.399617	mm,	Y =	678.826945	mm,	Z =	778.621701	mm,
	W =	-176.360249	deg,	P =	-59.752145	deg,	R =	40.936599	deg
};
P[601]{
   GP1:
	UF : 0, UT : 1,		CONFIG : 'N U T, 0, 0, 0',
	X =	2166.705364	mm,	Y =	671.355757	mm,	Z =	789.207706	mm,
	W =	-178.216172	deg,	P =	-61.753138	deg,	R =	39.811005	deg
};
P[602]{
   GP1:
	UF : 0, UT : 1,		CONFIG : 'N U T, 0, 0, 0',
	X =	2165.189236	mm,	Y =	665.743518	mm,	Z =	780.178079	mm,
	W =	143.046845	deg,	P =	-51.632346	deg,	R =	85.626215	deg
};
P[603]{
   GP1:
	UF : 0, UT : 1,		CONFIG : 'N U T, 0, 0, 0',
	X =	2150.343507	mm,	Y =	673.177312	mm,	Z =	769.483427	mm,
	W =	143.046845	deg,	P =	-51.632346	deg,	R =	85.626215	deg
};
P[604]{
   GP1:
	UF : 0, UT : 1,		CONFIG : 'N U T, 0, 0, 0',
	X =	2135.103492	mm,	Y =	679.818147	mm,	Z =	759.273692	mm,
	W =	145.481192	deg,	P =	-51.412420	deg,	R =	86.190140	deg
};
P[605]{
   GP1:
	UF : 0, UT : 1,		CONFIG : 'N U T, 0, 0, 0',
	X =	2119.195949	mm,	Y =	685.614735	mm,	Z =	749.659247	mm,
	W =	149.091816	deg,	P =	-50.236619	deg,	R =	85.968864	deg
};
P[606]{
   GP1:
	UF : 0, UT : 1,		CONFIG : 'N U T, 0, 0, 0',
	X =	2102.664262	mm,	Y =	690.434636	mm,	Z =	740.579534	mm,
	W =	152.358348	deg,	P =	-49.940332	deg,	R =	86.626468	deg
};
P[607]{
   GP1:
	UF : 0, UT : 1,		CONFIG : 'N U T, 0, 0, 0',
	X =	2085.562598	mm,	Y =	694.349940	mm,	Z =	732.146201	mm,
	W =	155.798072	deg,	P =	-49.144058	deg,	R =	86.848892	deg
};
P[608]{
   GP1:
	UF : 0, UT : 1,		CONFIG : 'N U T, 0, 0, 0',
	X =	2067.903936	mm,	Y =	696.910148	mm,	Z =	724.596298	mm,
	W =	160.268729	deg,	P =	-48.895303	deg,	R =	87.664943	deg
};
P[609]{
   GP1:
	UF : 0, UT : 1,		CONFIG : 'N U T, 0, 0, 0',
	X =	2049.759056	mm,	Y =	698.360716	mm,	Z =	717.805624	mm,
	W =	164.099329	deg,	P =	-49.167940	deg,	R =	88.449597	deg
};
P[610]{
   GP1:
	UF : 0, UT : 1,		CONFIG : 'N U T, 0, 0, 0',
	X =	2031.243271	mm,	Y =	698.446273	mm,	Z =	712.209431	mm,
	W =	169.217573	deg,	P =	-47.571614	deg,	R =	88.609921	deg
};
P[611]{
   GP1:
	UF : 0, UT : 1,		CONFIG : 'N U T, 0, 0, 0',
	X =	2012.496277	mm,	Y =	697.053284	mm,	Z =	707.605780	mm,
	W =	174.221494	deg,	P =	-47.899894	deg,	R =	89.273610	deg
};
P[612]{
   GP1:
	UF : 0, UT : 1,		CONFIG : 'N U T, 0, 0, 0',
	X =	1993.687234	mm,	Y =	694.166696	mm,	Z =	704.358636	mm,
	W =	179.800298	deg,	P =	-46.850562	deg,	R =	89.703076	deg
};
P[613]{
   GP1:
	UF : 0, UT : 1,		CONFIG : 'N U T, 0, 0, 0',
	X =	1974.892676	mm,	Y =	689.996246	mm,	Z =	702.146105	mm,
	W =	-175.501345	deg,	P =	-46.571460	deg,	R =	90.057240	deg
};
P[614]{
   GP1:
	UF : 0, UT : 1,		CONFIG : 'N U T, 0, 0, 0',
	X =	1956.445466	mm,	Y =	684.357805	mm,	Z =	701.228551	mm,
	W =	-169.681243	deg,	P =	-46.520650	deg,	R =	90.314120	deg
};
P[615]{
   GP1:
	UF : 0, UT : 1,		CONFIG : 'N U T, 0, 0, 0',
	X =	1938.271250	mm,	Y =	677.589423	mm,	Z =	701.357764	mm,
	W =	-164.921112	deg,	P =	-46.563556	deg,	R =	90.352997	deg
};
P[616]{
   GP1:
	UF : 0, UT : 1,		CONFIG : 'N U T, 0, 0, 0',
	X =	1920.644300	mm,	Y =	669.679951	mm,	Z =	702.675189	mm,
	W =	-160.042076	deg,	P =	-45.834095	deg,	R =	90.640523	deg
};
P[617]{
   GP1:
	UF : 0, UT : 1,		CONFIG : 'N U T, 0, 0, 0',
	X =	1903.513295	mm,	Y =	660.801919	mm,	Z =	704.924115	mm,
	W =	-155.766094	deg,	P =	-45.588606	deg,	R =	90.678500	deg
};
P[618]{
   GP1:
	UF : 0, UT : 1,		CONFIG : 'N U T, 0, 0, 0',
	X =	1886.981714	mm,	Y =	651.044052	mm,	Z =	708.021326	mm,
	W =	-151.126977	deg,	P =	-46.014088	deg,	R =	90.143614	deg
};
P[619]{
   GP1:
	UF : 0, UT : 1,		CONFIG : 'N U T, 0, 0, 0',
	X =	1871.066220	mm,	Y =	640.601575	mm,	Z =	712.051886	mm,
	W =	-147.954426	deg,	P =	-44.875463	deg,	R =	90.809532	deg
};
P[620]{
   GP1:
	UF : 0, UT : 1,		CONFIG : 'N U T, 0, 0, 0',
	X =	1855.782880	mm,	Y =	629.464477	mm,	Z =	716.760509	mm,
	W =	-144.421179	deg,	P =	-44.671006	deg,	R =	90.723472	deg
};
P[621]{
   GP1:
	UF : 0, UT : 1,		CONFIG : 'N U T, 0, 0, 0',
	X =	1841.125900	mm,	Y =	617.764322	mm,	Z =	722.129823	mm,
	W =	-141.106534	deg,	P =	-44.498035	deg,	R =	90.576842	deg
};
P[622]{
   GP1:
	UF : 0, UT : 1,		CONFIG : 'N U T, 0, 0, 0',
	X =	1827.014981	mm,	Y =	605.608957	mm,	Z =	728.049206	mm,
	W =	-138.260808	deg,	P =	-44.377018	deg,	R =	90.377442	deg
};
P[623]{
   GP1:
	UF : 0, UT : 1,		CONFIG : 'N U T, 0, 0, 0',
	X =	1830.186433	mm,	Y =	600.968014	mm,	Z =	719.641090	mm,
	W =	-127.565022	deg,	P =	-24.112506	deg,	R =	69.878322	deg
};
P[624]{
   GP1:
	UF : 0, UT : 1,		CONFIG : 'N U T, 0, 0, 0',
	X =	1844.406066	mm,	Y =	613.020734	mm,	Z =	713.783176	mm,
	W =	-127.565022	deg,	P =	-24.112506	deg,	R =	69.878322	deg
};
P[625]{
   GP1:
	UF : 0, UT : 1,		CONFIG : 'N U T, 0, 0, 0',
	X =	1859.060890	mm,	Y =	624.512660	mm,	Z =	708.531504	mm,
	W =	-129.106237	deg,	P =	-25.244701	deg,	R =	68.536125	deg
};
P[626]{
   GP1:
	UF : 0, UT : 1,		CONFIG : 'N U T, 0, 0, 0',
	X =	1874.351737	mm,	Y =	635.396368	mm,	Z =	704.034892	mm,
	W =	-131.566582	deg,	P =	-26.448976	deg,	R =	67.214384	deg
};
P[627]{
   GP1:
	UF : 0, UT : 1,		CONFIG : 'N U T, 0, 0, 0',
	X =	1890.235328	mm,	Y =	645.697210	mm,	Z =	700.211067	mm,
	W =	-133.933096	deg,	P =	-27.533446	deg,	R =	66.065185	deg
};
P[628]{
   GP1:
	UF : 0, UT : 1,		CONFIG : 'N U T, 0, 0, 0',
	X =	1906.685725	mm,	Y =	655.304708	mm,	Z =	697.195741	mm,
	W =	-137.055157	deg,	P =	-28.479981	deg,	R =	65.094462	deg
};
P[629]{
   GP1:
	UF : 0, UT : 1,		CONFIG : 'N U T, 0, 0, 0',
	X =	1923.752495	mm,	Y =	663.905655	mm,	Z =	695.063922	mm,
	W =	-139.126326	deg,	P =	-30.721245	deg,	R =	62.821235	deg
};
P[630]{
   GP1:
	UF : 0, UT : 1,		CONFIG : 'N U T, 0, 0, 0',
	X =	1941.315166	mm,	Y =	671.708774	mm,	Z =	693.922883	mm,
	W =	-142.712574	deg,	P =	-31.771969	deg,	R =	61.791548	deg
};
P[631]{
   GP1:
	UF : 0, UT : 1,		CONFIG : 'N U T, 0, 0, 0',
	X =	1959.343328	mm,	Y =	678.225394	mm,	Z =	693.894721	mm,
	W =	-145.817784	deg,	P =	-34.139676	deg,	R =	59.589837	deg
};
P[632]{
   GP1:
	UF : 0, UT : 1,		CONFIG : 'N U T, 0, 0, 0',
	X =	1977.713732	mm,	Y =	683.661111	mm,	Z =	695.038488	mm,
	W =	-150.289929	deg,	P =	-35.248214	deg,	R =	58.436771	deg
};
P[633]{
   GP1:
	UF : 0, UT : 1,		CONFIG : 'N U T, 0, 0, 0',
	X =	1996.312507	mm,	Y =	687.547618	mm,	Z =	697.306445	mm,
	W =	-152.727386	deg,	P =	-38.588970	deg,	R =	55.691088	deg
};
P[634]{
   GP1:
	UF : 0, UT : 1,		CONFIG : 'N U T, 0, 0, 0',
	X =	2014.974439	mm,	Y =	690.256118	mm,	Z =	700.785119	mm,
	W =	-156.779589	deg,	P =	-40.169764	deg,	R =	54.221824	deg
};
P[635]{
   GP1:
	UF : 0, UT : 1,		CONFIG : 'N U T, 0, 0, 0',
	X =	2033.504908	mm,	Y =	691.436687	mm,	Z =	705.412269	mm,
	W =	-160.165810	deg,	P =	-42.857182	deg,	R =	52.069950	deg
};
P[636]{
   GP1:
	UF : 0, UT : 1,		CONFIG : 'N U T, 0, 0, 0',
	X =	2051.889090	mm,	Y =	691.387478	mm,	Z =	710.980889	mm,
	W =	-162.556001	deg,	P =	-45.384755	deg,	R =	50.218562	deg
};
P[637]{
   GP1:
	UF : 0, UT : 1,		CONFIG : 'N U T, 0, 0, 0',
	X =	2069.673172	mm,	Y =	689.831492	mm,	Z =	717.798013	mm,
	W =	-167.096667	deg,	P =	-47.499449	deg,	R =	48.328229	deg
};
P[638]{
   GP1:
	UF : 0, UT : 1,		CONFIG : 'N U T, 0, 0, 0',
	X =	2087.197193	mm,	Y =	687.162692	mm,	Z =	725.327348	mm,
	W =	-169.266251	deg,	P =	-49.573136	deg,	R =	46.844442	deg
};
P[639]{
   GP1:
	UF : 0, UT : 1,		CONFIG : 'N U T, 0, 0, 0',
	X =	2104.136484	mm,	Y =	683.388061	mm,	Z =	733.626583	mm,
	W =	-171.732866	deg,	P =	-51.770179	deg,	R =	45.268279	deg
};
P[640]{
   GP1:
	UF : 0, UT : 1,		CONFIG : 'N U T, 0, 0, 0',
	X =	2120.397656	mm,	Y =	678.425684	mm,	Z =	742.608196	mm,
	W =	-173.322643	deg,	P =	-55.009169	deg,	R =	43.478437	deg
};
P[641]{
   GP1:
	UF : 0, UT : 1,		CONFIG : 'N U T, 0, 0, 0',
	X =	2136.130088	mm,	Y =	672.694339	mm,	Z =	752.217521	mm,
	W =	-175.534066	deg,	P =	-56.425118	deg,	R =	42.371327	deg
};
P[642]{
   GP1:
	UF : 0, UT : 1,		CONFIG : 'N U T, 0, 0, 0',
	X =	2151.203842	mm,	Y =	666.088044	mm,	Z =	762.279759	mm,
	W =	-177.115003	deg,	P =	-58.623100	deg,	R =	41.135298	deg
};
P[643]{
   GP1:
	UF : 0, UT : 1,		CONFIG : 'N U T, 0, 0, 0',
	X =	2165.684741	mm,	Y =	658.783005	mm,	Z =	772.805950	mm,
	W =	-178.909192	deg,	P =	-60.118232	deg,	R =	40.108237	deg
};
P[644]{
   GP1:
	UF : 0, UT : 1,		CONFIG : 'N U T, 0, 0, 0',
	X =	2162.115575	mm,	Y =	653.862524	mm,	Z =	762.439384	mm,
	W =	142.678808	deg,	P =	-51.719136	deg,	R =	85.612288	deg
};
P[645]{
   GP1:
	UF : 0, UT : 1,		CONFIG : 'N U T, 0, 0, 0',
	X =	2154.626979	mm,	Y =	657.679728	mm,	Z =	756.988137	mm,
	W =	142.678808	deg,	P =	-51.719136	deg,	R =	85.612288	deg
};
P[646]{
   GP1:
	UF : 0, UT : 1,		CONFIG : 'N U T, 0, 0, 0',
	X =	2139.413560	mm,	Y =	664.463085	mm,	Z =	746.779913	mm,
	W =	145.755458	deg,	P =	-50.489146	deg,	R =	85.100754	deg
};
P[647]{
   GP1:
	UF : 0, UT : 1,		CONFIG : 'N U T, 0, 0, 0',
	X =	2123.543386	mm,	Y =	670.432830	mm,	Z =	736.910224	mm,
	W =	148.315168	deg,	P =	-50.497381	deg,	R =	86.008267	deg
};
P[648]{
   GP1:
	UF : 0, UT : 1,		CONFIG : 'N U T, 0, 0, 0',
	X =	2107.045835	mm,	Y =	675.562139	mm,	Z =	727.698619	mm,
	W =	151.918187	deg,	P =	-49.126050	deg,	R =	85.750689	deg
};
P[649]{
   GP1:
	UF : 0, UT : 1,		CONFIG : 'N U T, 0, 0, 0',
	X =	2089.941003	mm,	Y =	679.583011	mm,	Z =	719.121619	mm,
	W =	155.510689	deg,	P =	-48.708680	deg,	R =	86.445687	deg
};
P[650]{
   GP1:
	UF : 0, UT : 1,		CONFIG : 'N U T, 0, 0, 0',
	X =	2072.261996	mm,	Y =	682.581685	mm,	Z =	711.361739	mm,
	W =	159.477147	deg,	P =	-47.019765	deg,	R =	86.384045	deg
};
P[651]{
   GP1:
	UF : 0, UT : 1,		CONFIG : 'N U T, 0, 0, 0',
	X =	2054.103279	mm,	Y =	684.176667	mm,	Z =	704.473284	mm,
	W =	163.831325	deg,	P =	-46.773832	deg,	R =	87.338981	deg
};
P[652]{
   GP1:
	UF : 0, UT : 1,		CONFIG : 'N U T, 0, 0, 0',
	X =	2035.535592	mm,	Y =	684.444888	mm,	Z =	698.591985	mm,
	W =	168.352013	deg,	P =	-46.417258	deg,	R =	88.135841	deg
};
P[653]{
   GP1:
	UF : 0, UT : 1,		CONFIG : 'N U T, 0, 0, 0',
	X =	2016.716138	mm,	Y =	683.285041	mm,	Z =	693.732509	mm,
	W =	173.189886	deg,	P =	-47.139457	deg,	R =	89.046410	deg
};
P[654]{
   GP1:
	UF : 0, UT : 1,		CONFIG : 'N U T, 0, 0, 0',
	X =	1997.753734	mm,	Y =	680.830957	mm,	Z =	690.154130	mm,
	W =	177.987903	deg,	P =	-45.399314	deg,	R =	89.500783	deg
};
P[655]{
   GP1:
	UF : 0, UT : 1,		CONFIG : 'N U T, 0, 0, 0',
	X =	1978.925728	mm,	Y =	676.719330	mm,	Z =	687.813015	mm,
	W =	-176.222276	deg,	P =	-45.580497	deg,	R =	90.129849	deg
};
P[656]{
   GP1:
	UF : 0, UT : 1,		CONFIG : 'N U T, 0, 0, 0',
	X =	1960.277800	mm,	Y =	671.277768	mm,	Z =	686.663272	mm,
	W =	-170.983913	deg,	P =	-45.731765	deg,	R =	90.469866	deg
};
P[657]{
   GP1:
	UF : 0, UT : 1,		CONFIG : 'N U T, 0, 0, 0',
	X =	1941.954660	mm,	Y =	664.654063	mm,	Z =	686.688571	mm,
	W =	-166.298991	deg,	P =	-45.084729	deg,	R =	90.885804	deg
};
P[658]{
   GP1:
	UF : 0, UT : 1,		CONFIG : 'N U T, 0, 0, 0',
	X =	1924.181000	mm,	Y =	656.765782	mm,	Z =	687.781954	mm,
	W =	-160.600005	deg,	P =	-45.992901	deg,	R =	90.568296	deg
};
P[659]{
   GP1:
	UF : 0, UT : 1,		CONFIG : 'N U T, 0, 0, 0',
	X =	1906.829146	mm,	Y =	648.049670	mm,	Z =	689.968893	mm,
	W =	-157.288636	deg,	P =	-44.416861	deg,	R =	91.408247	deg
};
P[660]{
   GP1:
	UF : 0, UT : 1,		CONFIG : 'N U T, 0, 0, 0',
	X =	1890.206371	mm,	Y =	638.299644	mm,	Z =	693.063133	mm,
	W =	-152.522973	deg,	P =	-44.497475	deg,	R =	91.306329	deg
};
P[661]{
   GP1:
	UF : 0, UT : 1,		CONFIG : 'N U T, 0, 0, 0',
	X =	1874.181745	mm,	Y =	627.795382	mm,	Z =	697.033454	mm,
	W =	-148.806570	deg,	P =	-44.117059	deg,	R =	91.473947	deg
};
P[662]{
   GP1:
	UF : 0, UT : 1,		CONFIG : 'N U T, 0, 0, 0',
	X =	1858.699458	mm,	Y =	616.680038	mm,	Z =	701.682410	mm,
	W =	-145.731016	deg,	P =	-43.850493	deg,	R =	91.558846	deg
};
P[663]{
   GP1:
	UF : 0, UT : 1,		CONFIG : 'N U T, 0, 0, 0',
	X =	1843.871555	mm,	Y =	604.980266	mm,	Z =	706.974182	mm,
	W =	-142.214650	deg,	P =	-43.924002	deg,	R =	91.256181	deg
};
P[664]{
   GP1:
	UF : 0, UT : 1,		CONFIG : 'N U T, 0, 0, 0',
	X =	1829.611996	mm,	Y =	592.837656	mm,	Z =	712.892226	mm,
	W =	-139.758988	deg,	P =	-43.374101	deg,	R =	91.622912	deg
};
P[665]{
   GP1:
	UF : 0, UT : 1,		CONFIG : 'N U T, 0, 0, 0',
	X =	1834.648759	mm,	Y =	589.541716	mm,	Z =	703.860764	mm,
	W =	-128.809927	deg,	P =	-24.025504	deg,	R =	70.058166	deg
};
P[666]{
   GP1:
	UF : 0, UT : 1,		CONFIG : 'N U T, 0, 0, 0',
	X =	1849.103589	mm,	Y =	601.516346	mm,	Z =	698.138987	mm,
	W =	-128.809927	deg,	P =	-24.025504	deg,	R =	70.058166	deg
};
P[667]{
   GP1:
	UF : 0, UT : 1,		CONFIG : 'N U T, 0, 0, 0',
	X =	1863.957521	mm,	Y =	612.980014	mm,	Z =	693.037549	mm,
	W =	-130.933824	deg,	P =	-24.740686	deg,	R =	69.238353	deg
};
P[668]{
   GP1:
	UF : 0, UT : 1,		CONFIG : 'N U T, 0, 0, 0',
	X =	1879.404203	mm,	Y =	623.847430	mm,	Z =	688.578732	mm,
	W =	-133.009448	deg,	P =	-25.905918	deg,	R =	67.895222	deg
};
P[669]{
   GP1:
	UF : 0, UT : 1,		CONFIG : 'N U T, 0, 0, 0',
	X =	1895.512762	mm,	Y =	633.942630	mm,	Z =	684.967489	mm,
	W =	-135.503209	deg,	P =	-27.454759	deg,	R =	66.183556	deg
};
P[670]{
   GP1:
	UF : 0, UT : 1,		CONFIG : 'N U T, 0, 0, 0',
	X =	1912.205249	mm,	Y =	643.363165	mm,	Z =	682.207273	mm,
	W =	-138.902265	deg,	P =	-28.255662	deg,	R =	65.309794	deg
};
P[671]{
   GP1:
	UF : 0, UT : 1,		CONFIG : 'N U T, 0, 0, 0',
	X =	1929.473008	mm,	Y =	651.849804	mm,	Z =	680.290285	mm,
	W =	-141.405074	deg,	P =	-29.980746	deg,	R =	63.522914	deg
};
P[672]{
   GP1:
	UF : 0, UT : 1,		CONFIG : 'N U T, 0, 0, 0',
	X =	1947.260634	mm,	Y =	659.233473	mm,	Z =	679.491129	mm,
	W =	-144.653927	deg,	P =	-31.920471	deg,	R =	61.590980	deg
};
P[673]{
   GP1:
	UF : 0, UT : 1,		CONFIG : 'N U T, 0, 0, 0',
	X =	1965.476747	mm,	Y =	665.616558	mm,	Z =	679.733828	mm,
	W =	-148.361140	deg,	P =	-33.194827	deg,	R =	60.260654	deg
};
P[674]{
   GP1:
	UF : 0, UT : 1,		CONFIG : 'N U T, 0, 0, 0',
	X =	1983.994085	mm,	Y =	670.565682	mm,	Z =	681.201468	mm,
	W =	-151.943364	deg,	P =	-35.585255	deg,	R =	58.035665	deg
};
P[675]{
   GP1:
	UF : 0, UT : 1,		CONFIG : 'N U T, 0, 0, 0',
	X =	2002.711943	mm,	Y =	674.312606	mm,	Z =	683.815068	mm,
	W =	-155.869664	deg,	P =	-37.127469	deg,	R =	56.461903	deg
};
P[676]{
   GP1:
	UF : 0, UT : 1,		CONFIG : 'N U T, 0, 0, 0',
	X =	2021.448057	mm,	Y =	676.504572	mm,	Z =	687.540374	mm,
	W =	-158.164255	deg,	P =	-40.572855	deg,	R =	53.797246	deg
};
P[677]{
   GP1:
	UF : 0, UT : 1,		CONFIG : 'N U T, 0, 0, 0',
	X =	2040.008674	mm,	Y =	677.385702	mm,	Z =	692.515832	mm,
	W =	-162.220360	deg,	P =	-42.438045	deg,	R =	52.050180	deg
};
P[678]{
   GP1:
	UF : 0, UT : 1,		CONFIG : 'N U T, 0, 0, 0',
	X =	2058.274831	mm,	Y =	676.836955	mm,	Z =	698.560080	mm,
	W =	-165.757084	deg,	P =	-44.645669	deg,	R =	50.143534	deg
};
P[679]{
   GP1:
	UF : 0, UT : 1,		CONFIG : 'N U T, 0, 0, 0',
	X =	2076.092190	mm,	Y =	674.913835	mm,	Z =	705.616897	mm,
	W =	-169.094812	deg,	P =	-46.883426	deg,	R =	48.248581	deg
};
P[680]{
   GP1:
	UF : 0, UT : 1,		CONFIG : 'N U T, 0, 0, 0',
	X =	2093.534757	mm,	Y =	671.920003	mm,	Z =	713.422690	mm,
	W =	-171.480340	deg,	P =	-48.754207	deg,	R =	46.748783	deg
};
P[681]{
   GP1:
	UF : 0, UT : 1,		CONFIG : 'N U T, 0, 0, 0',
	X =	2110.275365	mm,	Y =	667.616064	mm,	Z =	721.982737	mm,
	W =	-173.108336	deg,	P =	-52.282022	deg,	R =	44.711605	deg
};
P[682]{
   GP1:
	UF : 0, UT : 1,		CONFIG : 'N U T, 0, 0, 0',
	X =	2126.508931	mm,	Y =	662.408688	mm,	Z =	731.181789	mm,
	W =	-174.445271	deg,	P =	-54.833034	deg,	R =	43.286519	deg
};
P[683]{
   GP1:
	UF : 0, UT : 1,		CONFIG : 'N U T, 0, 0, 0',
	X =	2142.077885	mm,	Y =	656.417401	mm,	Z =	741.024271	mm,
	W =	-177.214153	deg,	P =	-55.867382	deg,	R =	42.097385	deg
};
P[684]{
   GP1:
	UF : 0, UT : 1,		CONFIG : 'N U T, 0, 0, 0',
	X =	2156.775071	mm,	Y =	649.653221	mm,	Z =	751.067006	mm,
	W =	-178.383503	deg,	P =	-58.281820	deg,	R =	40.869535	deg
};
P[685]{
   GP1:
	UF : 0, UT : 1,		CONFIG : 'N U T, 0, 0, 0',
	X =	2164.352728	mm,	Y =	645.951262	mm,	Z =	756.542682	mm,
	W =	-179.798253	deg,	P =	-58.505418	deg,	R =	40.305337	deg
};
P[686]{
   GP1:
	UF : 0, UT : 1,		CONFIG : 'N U T, 0, 0, 0',
	X =	2159.172357	mm,	Y =	641.516290	mm,	Z =	745.282120	mm,
	W =	145.223990	deg,	P =	-49.893982	deg,	R =	84.109476	deg
};
P[687]{
   GP1:
	UF : 0, UT : 1,		CONFIG : 'N U T, 0, 0, 0',
	X =	2144.078408	mm,	Y =	648.582105	mm,	Z =	734.822041	mm,
	W =	145.223990	deg,	P =	-49.893982	deg,	R =	84.109476	deg
};
P[688]{
   GP1:
	UF : 0, UT : 1,		CONFIG : 'N U T, 0, 0, 0',
	X =	2128.462028	mm,	Y =	654.684453	mm,	Z =	725.003295	mm,
	W =	148.524568	deg,	P =	-48.958814	deg,	R =	84.369735	deg
};
P[689]{
   GP1:
	UF : 0, UT : 1,		CONFIG : 'N U T, 0, 0, 0',
	X =	2112.232354	mm,	Y =	659.949703	mm,	Z =	715.679587	mm,
	W =	151.486790	deg,	P =	-48.328720	deg,	R =	84.859399	deg
};
P[690]{
   GP1:
	UF : 0, UT : 1,		CONFIG : 'N U T, 0, 0, 0',
	X =	2095.407290	mm,	Y =	664.326787	mm,	Z =	707.042791	mm,
	W =	155.087028	deg,	P =	-46.469774	deg,	R =	84.606417	deg
};
P[691]{
   GP1:
	UF : 0, UT : 1,		CONFIG : 'N U T, 0, 0, 0',
	X =	2078.018115	mm,	Y =	667.324785	mm,	Z =	699.094074	mm,
	W =	158.817660	deg,	P =	-47.302021	deg,	R =	86.374504	deg
};
P[692]{
   GP1:
	UF : 0, UT : 1,		CONFIG : 'N U T, 0, 0, 0',
	X =	2060.093875	mm,	Y =	669.488011	mm,	Z =	691.981133	mm,
	W =	162.368447	deg,	P =	-45.495816	deg,	R =	86.382082	deg
};
P[693]{
   GP1:
	UF : 0, UT : 1,		CONFIG : 'N U T, 0, 0, 0',
	X =	2041.814450	mm,	Y =	670.020604	mm,	Z =	685.872952	mm,
	W =	167.242747	deg,	P =	-45.884221	deg,	R =	87.748599	deg
};
P[694]{
   GP1:
	UF : 0, UT : 1,		CONFIG : 'N U T, 0, 0, 0',
	X =	2023.162097	mm,	Y =	669.382224	mm,	Z =	680.845092	mm,
	W =	171.537102	deg,	P =	-44.375930	deg,	R =	88.282388	deg
};
P[695]{
   GP1:
	UF : 0, UT : 1,		CONFIG : 'N U T, 0, 0, 0',
	X =	2004.406379	mm,	Y =	667.188755	mm,	Z =	676.995124	mm,
	W =	176.606817	deg,	P =	-43.719006	deg,	R =	89.218974	deg
};
P[696]{
   GP1:
	UF : 0, UT : 1,		CONFIG : 'N U T, 0, 0, 0',
	X =	1985.624134	mm,	Y =	663.648380	mm,	Z =	674.251279	mm,
	W =	-178.724914	deg,	P =	-43.426650	deg,	R =	90.027713	deg
};
P[697]{
   GP1:
	UF : 0, UT : 1,		CONFIG : 'N U T, 0, 0, 0',
	X =	1967.052199	mm,	Y =	658.671484	mm,	Z =	672.675445	mm,
	W =	-173.348718	deg,	P =	-44.158718	deg,	R =	90.635695	deg
};
P[698]{
   GP1:
	UF : 0, UT : 1,		CONFIG : 'N U T, 0, 0, 0',
	X =	1948.805178	mm,	Y =	652.420637	mm,	Z =	672.376486	mm,
	W =	-168.250669	deg,	P =	-43.781936	deg,	R =	91.213878	deg
};
P[699]{
   GP1:
	UF : 0, UT : 1,		CONFIG : 'N U T, 0, 0, 0',
	X =	1930.944876	mm,	Y =	645.039921	mm,	Z =	673.144147	mm,
	W =	-163.724385	deg,	P =	-43.548559	deg,	R =	91.633832	deg
};
P[700]{
   GP1:
	UF : 0, UT : 1,		CONFIG : 'N U T, 0, 0, 0',
	X =	1913.673326	mm,	Y =	636.574810	mm,	Z =	675.041531	mm,
	W =	-159.230135	deg,	P =	-42.864791	deg,	R =	92.234828	deg
};
P[701]{
   GP1:
	UF : 0, UT : 1,		CONFIG : 'N U T, 0, 0, 0',
	X =	1896.943666	mm,	Y =	627.169425	mm,	Z =	677.787219	mm,
	W =	-154.834119	deg,	P =	-43.357065	deg,	R =	92.095946	deg
};
P[702]{
   GP1:
	UF : 0, UT : 1,		CONFIG : 'N U T, 0, 0, 0',
	X =	1880.759159	mm,	Y =	617.060231	mm,	Z =	681.391364	mm,
	W =	-151.429408	deg,	P =	-42.930970	deg,	R =	92.439373	deg
};
P[703]{
   GP1:
	UF : 0, UT : 1,		CONFIG : 'N U T, 0, 0, 0',
	X =	1865.278422	mm,	Y =	606.200017	mm,	Z =	685.772722	mm,
	W =	-147.410223	deg,	P =	-43.048816	deg,	R =	92.322386	deg
};
P[704]{
   GP1:
	UF : 0, UT : 1,		CONFIG : 'N U T, 0, 0, 0',
	X =	1850.328656	mm,	Y =	594.804681	mm,	Z =	690.829294	mm,
	W =	-144.582387	deg,	P =	-42.722355	deg,	R =	92.547138	deg
};
P[705]{
   GP1:
	UF : 0, UT : 1,		CONFIG : 'N U T, 0, 0, 0',
	X =	1836.004133	mm,	Y =	582.899310	mm,	Z =	696.497233	mm,
	W =	-141.722044	deg,	P =	-42.432032	deg,	R =	92.733479	deg
};
P[706]{
   GP1:
	UF : 0, UT : 1,		CONFIG : 'N U T, 0, 0, 0',
	X =	1837.249416	mm,	Y =	576.031722	mm,	Z =	689.301689	mm,
	W =	-129.561461	deg,	P =	-23.198251	deg,	R =	71.142147	deg
};
P[707]{
   GP1:
	UF : 0, UT : 1,		CONFIG : 'N U T, 0, 0, 0',
	X =	1844.537667	mm,	Y =	582.170980	mm,	Z =	686.331440	mm,
	W =	-129.561461	deg,	P =	-23.198251	deg,	R =	71.142147	deg
};
P[708]{
   GP1:
	UF : 0, UT : 1,		CONFIG : 'N U T, 0, 0, 0',
	X =	1851.933727	mm,	Y =	588.141658	mm,	Z =	683.539003	mm,
	W =	-130.431559	deg,	P =	-23.792532	deg,	R =	70.401496	deg
};
P[709]{
   GP1:
	UF : 0, UT : 1,		CONFIG : 'N U T, 0, 0, 0',
	X =	1859.463321	mm,	Y =	594.028135	mm,	Z =	680.916087	mm,
	W =	-131.770195	deg,	P =	-24.007381	deg,	R =	70.146849	deg
};
P[710]{
   GP1:
	UF : 0, UT : 1,		CONFIG : 'N U T, 0, 0, 0',
	X =	1875.019720	mm,	Y =	605.366507	mm,	Z =	676.167793	mm,
	W =	-134.145193	deg,	P =	-24.411627	deg,	R =	69.634809	deg
};
P[711]{
   GP1:
	UF : 0, UT : 1,		CONFIG : 'N U T, 0, 0, 0',
	X =	1891.176199	mm,	Y =	615.996196	mm,	Z =	672.098431	mm,
	W =	-136.105531	deg,	P =	-25.776103	deg,	R =	68.027899	deg
};
P[712]{
   GP1:
	UF : 0, UT : 1,		CONFIG : 'N U T, 0, 0, 0',
	X =	1907.964737	mm,	Y =	625.842448	mm,	Z =	668.964799	mm,
	W =	-139.256187	deg,	P =	-26.942130	deg,	R =	66.654757	deg
};
P[713]{
   GP1:
	UF : 0, UT : 1,		CONFIG : 'N U T, 0, 0, 0',
	X =	1925.399079	mm,	Y =	634.729857	mm,	Z =	666.703103	mm,
	W =	-141.273689	deg,	P =	-29.048411	deg,	R =	64.435972	deg
};
P[714]{
   GP1:
	UF : 0, UT : 1,		CONFIG : 'N U T, 0, 0, 0',
	X =	1943.355828	mm,	Y =	642.708224	mm,	Z =	665.552517	mm,
	W =	-145.227649	deg,	P =	-30.075091	deg,	R =	63.227520	deg
};
P[715]{
   GP1:
	UF : 0, UT : 1,		CONFIG : 'N U T, 0, 0, 0',
	X =	1961.816369	mm,	Y =	649.376024	mm,	Z =	665.529176	mm,
	W =	-148.354409	deg,	P =	-32.355033	deg,	R =	60.968995	deg
};
P[716]{
   GP1:
	UF : 0, UT : 1,		CONFIG : 'N U T, 0, 0, 0',
	X =	1980.622177	mm,	Y =	654.916502	mm,	Z =	666.724525	mm,
	W =	-152.898563	deg,	P =	-33.355695	deg,	R =	59.661069	deg
};
P[717]{
   GP1:
	UF : 0, UT : 1,		CONFIG : 'N U T, 0, 0, 0',
	X =	1999.666742	mm,	Y =	659.018385	mm,	Z =	669.053627	mm,
	W =	-156.198445	deg,	P =	-35.652411	deg,	R =	57.478253	deg
};
P[718]{
   GP1:
	UF : 0, UT : 1,		CONFIG : 'N U T, 0, 0, 0',
	X =	2018.735985	mm,	Y =	661.561667	mm,	Z =	672.679118	mm,
	W =	-159.535257	deg,	P =	-38.478914	deg,	R =	55.005573	deg
};
P[719]{
   GP1:
	UF : 0, UT : 1,		CONFIG : 'N U T, 0, 0, 0',
	X =	2037.704377	mm,	Y =	662.678247	mm,	Z =	677.519063	mm,
	W =	-163.032867	deg,	P =	-40.800056	deg,	R =	52.915975	deg
};
P[720]{
   GP1:
	UF : 0, UT : 1,		CONFIG : 'N U T, 0, 0, 0',
	X =	2056.368023	mm,	Y =	662.315147	mm,	Z =	683.517680	mm,
	W =	-166.550838	deg,	P =	-43.152168	deg,	R =	50.822312	deg
};
P[721]{
   GP1:
	UF : 0, UT : 1,		CONFIG : 'N U T, 0, 0, 0',
	X =	2074.712671	mm,	Y =	660.598001	mm,	Z =	690.390023	mm,
	W =	-168.163425	deg,	P =	-46.454693	deg,	R =	48.675242	deg
};
P[722]{
   GP1:
	UF : 0, UT : 1,		CONFIG : 'N U T, 0, 0, 0',
	X =	2092.419680	mm,	Y =	657.654475	mm,	Z =	698.349706	mm,
	W =	-172.064871	deg,	P =	-48.026363	deg,	R =	46.943504	deg
};
P[723]{
   GP1:
	UF : 0, UT : 1,		CONFIG : 'N U T, 0, 0, 0',
	X =	2109.625276	mm,	Y =	653.454836	mm,	Z =	706.974713	mm,
	W =	-173.518294	deg,	P =	-51.088620	deg,	R =	45.134227	deg
};
P[724]{
   GP1:
	UF : 0, UT : 1,		CONFIG : 'N U T, 0, 0, 0',
	X =	2126.189322	mm,	Y =	648.298405	mm,	Z =	716.342284	mm,
	W =	-175.896730	deg,	P =	-52.938234	deg,	R =	43.651545	deg
};
P[725]{
   GP1:
	UF : 0, UT : 1,		CONFIG : 'N U T, 0, 0, 0',
	X =	2142.068872	mm,	Y =	642.137558	mm,	Z =	726.263862	mm,
	W =	-177.517490	deg,	P =	-55.408627	deg,	R =	42.168825	deg
};
P[726]{
   GP1:
	UF : 0, UT : 1,		CONFIG : 'N U T, 0, 0, 0',
	X =	2157.436425	mm,	Y =	635.325313	mm,	Z =	736.741680	mm,
	W =	-179.889010	deg,	P =	-55.970066	deg,	R =	41.097421	deg
};
P[727]{
   GP1:
	UF : 0, UT : 1,		CONFIG : 'N U T, 0, 0, 0',
	X =	2155.760498	mm,	Y =	628.862551	mm,	Z =	728.272871	mm,
	W =	147.220499	deg,	P =	-47.875155	deg,	R =	82.539063	deg
};
P[728]{
   GP1:
	UF : 0, UT : 1,		CONFIG : 'N U T, 0, 0, 0',
	X =	2140.369386	mm,	Y =	635.622413	mm,	Z =	717.980668	mm,
	W =	147.220499	deg,	P =	-47.875155	deg,	R =	82.539063	deg
};
P[729]{
   GP1:
	UF : 0, UT : 1,		CONFIG : 'N U T, 0, 0, 0',
	X =	2124.574656	mm,	Y =	641.521315	mm,	Z =	708.156680	mm,
	W =	149.352575	deg,	P =	-48.211078	deg,	R =	83.904349	deg
};
P[730]{
   GP1:
	UF : 0, UT : 1,		CONFIG : 'N U T, 0, 0, 0',
	X =	2108.135234	mm,	Y =	646.494687	mm,	Z =	699.041332	mm,
	W =	152.846319	deg,	P =	-47.161663	deg,	R =	84.316005	deg
};
P[731]{
   GP1:
	UF : 0, UT : 1,		CONFIG : 'N U T, 0, 0, 0',
	X =	2091.109387	mm,	Y =	650.684539	mm,	Z =	690.569056	mm,
	W =	156.214397	deg,	P =	-44.694164	deg,	R =	83.761180	deg
};
P[732]{
   GP1:
	UF : 0, UT : 1,		CONFIG : 'N U T, 0, 0, 0',
	X =	2073.529753	mm,	Y =	653.312303	mm,	Z =	682.897225	mm,
	W =	160.355007	deg,	P =	-45.146954	deg,	R =	85.587437	deg
};
P[733]{
   GP1:
	UF : 0, UT : 1,		CONFIG : 'N U T, 0, 0, 0',
	X =	2055.419632	mm,	Y =	654.944384	mm,	Z =	676.083048	mm,
	W =	163.995969	deg,	P =	-44.135840	deg,	R =	86.263226	deg
};
P[734]{
   GP1:
	UF : 0, UT : 1,		CONFIG : 'N U T, 0, 0, 0',
	X =	2036.959679	mm,	Y =	655.233619	mm,	Z =	670.197747	mm,
	W =	168.164042	deg,	P =	-43.971732	deg,	R =	87.388270	deg
};
P[735]{
   GP1:
	UF : 0, UT : 1,		CONFIG : 'N U T, 0, 0, 0',
	X =	2018.275464	mm,	Y =	653.914498	mm,	Z =	665.593849	mm,
	W =	173.488377	deg,	P =	-43.603484	deg,	R =	88.579875	deg
};
P[736]{
   GP1:
	UF : 0, UT : 1,		CONFIG : 'N U T, 0, 0, 0',
	X =	1999.409115	mm,	Y =	651.332959	mm,	Z =	662.127413	mm,
	W =	177.800963	deg,	P =	-42.160330	deg,	R =	89.415533	deg
};
P[737]{
   GP1:
	UF : 0, UT : 1,		CONFIG : 'N U T, 0, 0, 0',
	X =	1980.669157	mm,	Y =	647.231322	mm,	Z =	659.834399	mm,
	W =	-177.135413	deg,	P =	-42.133565	deg,	R =	90.418549	deg
};
P[738]{
   GP1:
	UF : 0, UT : 1,		CONFIG : 'N U T, 0, 0, 0',
	X =	1962.128308	mm,	Y =	641.822620	mm,	Z =	658.684426	mm,
	W =	-172.276900	deg,	P =	-42.398041	deg,	R =	91.149338	deg
};
P[739]{
   GP1:
	UF : 0, UT : 1,		CONFIG : 'N U T, 0, 0, 0',
	X =	1943.941789	mm,	Y =	635.191375	mm,	Z =	658.683297	mm,
	W =	-167.434762	deg,	P =	-42.537982	deg,	R =	91.712524	deg
};
P[740]{
   GP1:
	UF : 0, UT : 1,		CONFIG : 'N U T, 0, 0, 0',
	X =	1926.279262	mm,	Y =	627.389697	mm,	Z =	659.900305	mm,
	W =	-162.751570	deg,	P =	-41.872411	deg,	R =	92.469971	deg
};
P[741]{
   GP1:
	UF : 0, UT : 1,		CONFIG : 'N U T, 0, 0, 0',
	X =	1909.133015	mm,	Y =	618.574598	mm,	Z =	662.085713	mm,
	W =	-158.551834	deg,	P =	-41.761187	deg,	R =	92.900264	deg
};
P[742]{
   GP1:
	UF : 0, UT : 1,		CONFIG : 'N U T, 0, 0, 0',
	X =	1892.531740	mm,	Y =	608.904396	mm,	Z =	665.085352	mm,
	W =	-154.371405	deg,	P =	-42.390480	deg,	R =	92.754595	deg
};
P[743]{
   GP1:
	UF : 0, UT : 1,		CONFIG : 'N U T, 0, 0, 0',
	X =	1876.551771	mm,	Y =	598.519233	mm,	Z =	668.964633	mm,
	W =	-150.744700	deg,	P =	-42.124889	deg,	R =	93.065728	deg
};
P[744]{
   GP1:
	UF : 0, UT : 1,		CONFIG : 'N U T, 0, 0, 0',
	X =	1861.262310	mm,	Y =	587.454849	mm,	Z =	673.674519	mm,
	W =	-147.543295	deg,	P =	-41.399742	deg,	R =	93.747126	deg
};
P[745]{
   GP1:
	UF : 0, UT : 1,		CONFIG : 'N U T, 0, 0, 0',
	X =	1846.683459	mm,	Y =	575.895317	mm,	Z =	678.906871	mm,
	W =	-144.219076	deg,	P =	-41.748440	deg,	R =	93.467951	deg
};
P[746]{
   GP1:
	UF : 0, UT : 1,		CONFIG : 'N U T, 0, 0, 0',
	X =	1839.423088	mm,	Y =	569.830311	mm,	Z =	681.823923	mm,
	W =	-142.521290	deg,	P =	-41.376023	deg,	R =	93.832001	deg
};
P[747]{
   GP1:
	UF : 0, UT : 1,		CONFIG : 'N U T, 0, 0, 0',
	X =	1840.770818	mm,	Y =	562.839042	mm,	Z =	674.839583	mm,
	W =	-131.445954	deg,	P =	-22.130930	deg,	R =	72.495808	deg
};
P[748]{
   GP1:
	UF : 0, UT : 1,		CONFIG : 'N U T, 0, 0, 0',
	X =	1847.869129	mm,	Y =	568.816506	mm,	Z =	671.948221	mm,
	W =	-131.445954	deg,	P =	-22.130930	deg,	R =	72.495808	deg
};
P[749]{
   GP1:
	UF : 0, UT : 1,		CONFIG : 'N U T, 0, 0, 0',
	X =	1862.523070	mm,	Y =	580.304959	mm,	Z =	666.638463	mm,
	W =	-132.261945	deg,	P =	-23.403926	deg,	R =	70.882901	deg
};
P[750]{
   GP1:
	UF : 0, UT : 1,		CONFIG : 'N U T, 0, 0, 0',
	X =	1877.735773	mm,	Y =	591.229281	mm,	Z =	662.084860	mm,
	W =	-134.634207	deg,	P =	-24.432898	deg,	R =	69.596417	deg
};
P[751]{
   GP1:
	UF : 0, UT : 1,		CONFIG : 'N U T, 0, 0, 0',
	X =	1893.554691	mm,	Y =	601.536769	mm,	Z =	658.282978	mm,
	W =	-137.579549	deg,	P =	-25.249158	deg,	R =	68.549085	deg
};
P[752]{
   GP1:
	UF : 0, UT : 1,		CONFIG : 'N U T, 0, 0, 0',
	X =	1909.963817	mm,	Y =	611.124426	mm,	Z =	655.229164	mm,
	W =	-140.267287	deg,	P =	-26.341106	deg,	R =	67.217280	deg
};
P[753]{
   GP1:
	UF : 0, UT : 1,		CONFIG : 'N U T, 0, 0, 0',
	X =	1926.939827	mm,	Y =	619.865277	mm,	Z =	653.067525	mm,
	W =	-143.294623	deg,	P =	-27.602297	deg,	R =	65.711654	deg
};
P[754]{
   GP1:
	UF : 0, UT : 1,		CONFIG : 'N U T, 0, 0, 0',
	X =	1944.453099	mm,	Y =	627.617857	mm,	Z =	651.867147	mm,
	W =	-146.209342	deg,	P =	-29.274112	deg,	R =	63.867227	deg
};
P[755]{
   GP1:
	UF : 0, UT : 1,		CONFIG : 'N U T, 0, 0, 0',
	X =	1962.420554	mm,	Y =	634.220848	mm,	Z =	651.829749	mm,
	W =	-150.008801	deg,	P =	-30.886738	deg,	R =	62.028425	deg
};
P[756]{
   GP1:
	UF : 0, UT : 1,		CONFIG : 'N U T, 0, 0, 0',
	X =	1980.765232	mm,	Y =	639.593561	mm,	Z =	652.889374	mm,
	W =	-153.282576	deg,	P =	-32.894466	deg,	R =	59.967275	deg
};
P[757]{
   GP1:
	UF : 0, UT : 1,		CONFIG : 'N U T, 0, 0, 0',
	X =	1999.314901	mm,	Y =	643.592583	mm,	Z =	655.170222	mm,
	W =	-156.799886	deg,	P =	-35.168876	deg,	R =	57.733174	deg
};
P[758]{
   GP1:
	UF : 0, UT : 1,		CONFIG : 'N U T, 0, 0, 0',
	X =	2017.921761	mm,	Y =	646.255377	mm,	Z =	658.658172	mm,
	W =	-160.807447	deg,	P =	-36.922990	deg,	R =	55.807868	deg
};
P[759]{
   GP1:
	UF : 0, UT : 1,		CONFIG : 'N U T, 0, 0, 0',
	X =	2036.461984	mm,	Y =	647.576152	mm,	Z =	663.218474	mm,
	W =	-164.281400	deg,	P =	-38.845035	deg,	R =	53.850316	deg
};
P[760]{
   GP1:
	UF : 0, UT : 1,		CONFIG : 'N U T, 0, 0, 0',
	X =	2054.765935	mm,	Y =	647.405241	mm,	Z =	668.783506	mm,
	W =	-166.242152	deg,	P =	-42.376121	deg,	R =	51.329321	deg
};
P[761]{
   GP1:
	UF : 0, UT : 1,		CONFIG : 'N U T, 0, 0, 0',
	X =	2072.572868	mm,	Y =	645.958695	mm,	Z =	675.571894	mm,
	W =	-170.825235	deg,	P =	-43.641140	deg,	R =	49.467315	deg
};
P[762]{
   GP1:
	UF : 0, UT : 1,		CONFIG : 'N U T, 0, 0, 0',
	X =	2090.081449	mm,	Y =	643.265588	mm,	Z =	683.013571	mm,
	W =	-172.129932	deg,	P =	-46.632488	deg,	R =	47.595158	deg
};
P[763]{
   GP1:
	UF : 0, UT : 1,		CONFIG : 'N U T, 0, 0, 0',
	X =	2106.971628	mm,	Y =	639.460628	mm,	Z =	691.280647	mm,
	W =	-174.240061	deg,	P =	-49.273904	deg,	R =	45.732925	deg
};
P[764]{
   GP1:
	UF : 0, UT : 1,		CONFIG : 'N U T, 0, 0, 0',
	X =	2123.219911	mm,	Y =	634.572580	mm,	Z =	700.273536	mm,
	W =	-176.299041	deg,	P =	-51.759414	deg,	R =	44.001758	deg
};
P[765]{
   GP1:
	UF : 0, UT : 1,		CONFIG : 'N U T, 0, 0, 0',
	X =	2138.967075	mm,	Y =	628.937800	mm,	Z =	709.863744	mm,
	W =	-178.739118	deg,	P =	-52.601069	deg,	R =	42.770343	deg
};
P[766]{
   GP1:
	UF : 0, UT : 1,		CONFIG : 'N U T, 0, 0, 0',
	X =	2154.021998	mm,	Y =	622.290149	mm,	Z =	719.848310	mm,
	W =	-179.522474	deg,	P =	-55.809394	deg,	R =	41.299080	deg
};
P[767]{
   GP1:
	UF : 0, UT : 1,		CONFIG : 'N U T, 0, 0, 0',
	X =	2152.275255	mm,	Y =	615.685562	mm,	Z =	711.560006	mm,
	W =	148.311548	deg,	P =	-47.005797	deg,	R =	82.108329	deg
};
P[768]{
   GP1:
	UF : 0, UT : 1,		CONFIG : 'N U T, 0, 0, 0',
	X =	2136.659225	mm,	Y =	622.221251	mm,	Z =	701.388592	mm,
	W =	148.311548	deg,	P =	-47.005797	deg,	R =	82.108329	deg
};
P[769]{
   GP1:
	UF : 0, UT : 1,		CONFIG : 'N U T, 0, 0, 0',
	X =	2120.671055	mm,	Y =	627.924297	mm,	Z =	691.757632	mm,
	W =	150.731210	deg,	P =	-46.535642	deg,	R =	82.829288	deg
};
P[770]{
   GP1:
	UF : 0, UT : 1,		CONFIG : 'N U T, 0, 0, 0',
	X =	2104.038562	mm,	Y =	632.541257	mm,	Z =	682.796891	mm,
	W =	154.074842	deg,	P =	-46.215808	deg,	R =	84.014656	deg
};
P[771]{
   GP1:
	UF : 0, UT : 1,		CONFIG : 'N U T, 0, 0, 0',
	X =	2086.803450	mm,	Y =	636.328560	mm,	Z =	674.565248	mm,
	W =	157.509496	deg,	P =	-43.984723	deg,	R =	83.836511	deg
};
P[772]{
   GP1:
	UF : 0, UT : 1,		CONFIG : 'N U T, 0, 0, 0',
	X =	2069.025611	mm,	Y =	638.761886	mm,	Z =	667.209838	mm,
	W =	161.604981	deg,	P =	-42.380940	deg,	R =	84.640261	deg
};
P[773]{
   GP1:
	UF : 0, UT : 1,		CONFIG : 'N U T, 0, 0, 0',
	X =	2050.780031	mm,	Y =	639.823760	mm,	Z =	660.699167	mm,
	W =	165.565892	deg,	P =	-42.561561	deg,	R =	86.171957	deg
};
P[774]{
   GP1:
	UF : 0, UT : 1,		CONFIG : 'N U T, 0, 0, 0',
	X =	2032.183164	mm,	Y =	639.649559	mm,	Z =	655.209462	mm,
	W =	169.638369	deg,	P =	-41.910371	deg,	R =	87.283611	deg
};
P[775]{
   GP1:
	UF : 0, UT : 1,		CONFIG : 'N U T, 0, 0, 0',
	X =	2013.393427	mm,	Y =	638.062521	mm,	Z =	650.766246	mm,
	W =	174.117255	deg,	P =	-42.113889	deg,	R =	88.552854	deg
};
P[776]{
   GP1:
	UF : 0, UT : 1,		CONFIG : 'N U T, 0, 0, 0',
	X =	1994.585924	mm,	Y =	634.963415	mm,	Z =	647.639991	mm,
	W =	179.267856	deg,	P =	-41.665264	deg,	R =	89.740127	deg
};
P[777]{
   GP1:
	UF : 0, UT : 1,		CONFIG : 'N U T, 0, 0, 0',
	X =	1975.860484	mm,	Y =	630.468364	mm,	Z =	645.682640	mm,
	W =	-175.868001	deg,	P =	-41.699432	deg,	R =	90.705534	deg
};
P[778]{
   GP1:
	UF : 0, UT : 1,		CONFIG : 'N U T, 0, 0, 0',
	X =	1957.391598	mm,	Y =	624.686930	mm,	Z =	644.931566	mm,
	W =	-171.169691	deg,	P =	-41.291688	deg,	R =	91.593678	deg
};
P[779]{
   GP1:
	UF : 0, UT : 1,		CONFIG : 'N U T, 0, 0, 0',
	X =	1939.401239	mm,	Y =	617.571186	mm,	Z =	645.392328	mm,
	W =	-166.005315	deg,	P =	-41.411934	deg,	R =	92.299360	deg
};
P[780]{
   GP1:
	UF : 0, UT : 1,		CONFIG : 'N U T, 0, 0, 0',
	X =	1921.876414	mm,	Y =	609.389225	mm,	Z =	646.945477	mm,
	W =	-161.674027	deg,	P =	-41.119172	deg,	R =	92.947868	deg
};
P[781]{
   GP1:
	UF : 0, UT : 1,		CONFIG : 'N U T, 0, 0, 0',
	X =	1904.895665	mm,	Y =	600.272436	mm,	Z =	649.439691	mm,
	W =	-157.693318	deg,	P =	-41.006210	deg,	R =	93.417450	deg
};
P[782]{
   GP1:
	UF : 0, UT : 1,		CONFIG : 'N U T, 0, 0, 0',
	X =	1888.500888	mm,	Y =	590.346033	mm,	Z =	652.806493	mm,
	W =	-154.051806	deg,	P =	-40.793578	deg,	R =	93.870495	deg
};
P[783]{
   GP1:
	UF : 0, UT : 1,		CONFIG : 'N U T, 0, 0, 0',
	X =	1872.801362	mm,	Y =	579.657849	mm,	Z =	657.038600	mm,
	W =	-150.462851	deg,	P =	-40.421020	deg,	R =	94.419329	deg
};
P[784]{
   GP1:
	UF : 0, UT : 1,		CONFIG : 'N U T, 0, 0, 0',
	X =	1857.646394	mm,	Y =	568.365497	mm,	Z =	661.931423	mm,
	W =	-147.538508	deg,	P =	-40.297888	deg,	R =	94.713035	deg
};
P[785]{
   GP1:
	UF : 0, UT : 1,		CONFIG : 'N U T, 0, 0, 0',
	X =	1843.156152	mm,	Y =	556.511670	mm,	Z =	667.429545	mm,
	W =	-144.083249	deg,	P =	-40.722700	deg,	R =	94.466110	deg
};
P[786]{
   GP1:
	UF : 0, UT : 1,		CONFIG : 'N U T, 0, 0, 0',
	X =	1846.882922	mm,	Y =	551.328742	mm,	Z =	659.680152	mm,
	W =	-133.734918	deg,	P =	-22.065318	deg,	R =	72.469081	deg
};
P[787]{
   GP1:
	UF : 0, UT : 1,		CONFIG : 'N U T, 0, 0, 0',
	X =	1861.784941	mm,	Y =	563.253424	mm,	Z =	654.134357	mm,
	W =	-133.734918	deg,	P =	-22.065318	deg,	R =	72.469081	deg
};
P[788]{
   GP1:
	UF : 0, UT : 1,		CONFIG : 'N U T, 0, 0, 0',
	X =	1877.163992	mm,	Y =	574.506743	mm,	Z =	649.319365	mm,
	W =	-135.726387	deg,	P =	-23.199740	deg,	R =	70.979055	deg
};
P[789]{
   GP1:
	UF : 0, UT : 1,		CONFIG : 'N U T, 0, 0, 0',
	X =	1893.183189	mm,	Y =	585.106340	mm,	Z =	645.264263	mm,
	W =	-138.072299	deg,	P =	-24.406816	deg,	R =	69.441947	deg
};
P[790]{
   GP1:
	UF : 0, UT : 1,		CONFIG : 'N U T, 0, 0, 0',
	X =	1909.847353	mm,	Y =	594.921059	mm,	Z =	642.098894	mm,
	W =	-141.004223	deg,	P =	-25.623453	deg,	R =	67.897678	deg
};
P[791]{
   GP1:
	UF : 0, UT : 1,		CONFIG : 'N U T, 0, 0, 0',
	X =	1927.108206	mm,	Y =	603.908350	mm,	Z =	639.831353	mm,
	W =	-144.148719	deg,	P =	-26.726981	deg,	R =	66.471230	deg
};
P[792]{
   GP1:
	UF : 0, UT : 1,		CONFIG : 'N U T, 0, 0, 0',
	X =	1944.928720	mm,	Y =	611.864920	mm,	Z =	638.560598	mm,
	W =	-147.193392	deg,	P =	-28.346109	deg,	R =	64.593014	deg
};
P[793]{
   GP1:
	UF : 0, UT : 1,		CONFIG : 'N U T, 0, 0, 0',
	X =	1963.217644	mm,	Y =	618.717493	mm,	Z =	638.421509	mm,
	W =	-150.970699	deg,	P =	-29.724647	deg,	R =	62.863801	deg
};
P[794]{
   GP1:
	UF : 0, UT : 1,		CONFIG : 'N U T, 0, 0, 0',
	X =	1981.898212	mm,	Y =	624.174340	mm,	Z =	639.489270	mm,
	W =	-154.273617	deg,	P =	-32.085700	deg,	R =	60.439855	deg
};
P[795]{
   GP1:
	UF : 0, UT : 1,		CONFIG : 'N U T, 0, 0, 0',
	X =	2000.820314	mm,	Y =	628.340567	mm,	Z =	641.759413	mm,
	W =	-157.801899	deg,	P =	-34.049568	deg,	R =	58.357855	deg
};
P[796]{
   GP1:
	UF : 0, UT : 1,		CONFIG : 'N U T, 0, 0, 0',
	X =	2019.769262	mm,	Y =	630.919252	mm,	Z =	645.344909	mm,
	W =	-161.417181	deg,	P =	-36.700790	deg,	R =	55.829591	deg
};
P[797]{
   GP1:
	UF : 0, UT : 1,		CONFIG : 'N U T, 0, 0, 0',
	X =	2038.641005	mm,	Y =	632.110604	mm,	Z =	650.107096	mm,
	W =	-164.936777	deg,	P =	-38.797981	deg,	R =	53.724932	deg
};
P[798]{
   GP1:
	UF : 0, UT : 1,		CONFIG : 'N U T, 0, 0, 0',
	X =	2057.192655	mm,	Y =	631.795875	mm,	Z =	656.029244	mm,
	W =	-168.423330	deg,	P =	-41.183375	deg,	R =	51.456207	deg
};
P[799]{
   GP1:
	UF : 0, UT : 1,		CONFIG : 'N U T, 0, 0, 0',
	X =	2075.401408	mm,	Y =	630.157318	mm,	Z =	662.913931	mm,
	W =	-171.087882	deg,	P =	-43.584083	deg,	R =	49.418473	deg
};
P[800]{
   GP1:
	UF : 0, UT : 1,		CONFIG : 'N U T, 0, 0, 0',
	X =	2093.223494	mm,	Y =	627.449275	mm,	Z =	670.585125	mm,
	W =	-173.350554	deg,	P =	-45.507941	deg,	R =	47.758153	deg
};
P[801]{
   GP1:
	UF : 0, UT : 1,		CONFIG : 'N U T, 0, 0, 0',
	X =	2110.268253	mm,	Y =	623.380084	mm,	Z =	679.172780	mm,
	W =	-176.156027	deg,	P =	-48.150098	deg,	R =	45.575683	deg
};
P[802]{
   GP1:
	UF : 0, UT : 1,		CONFIG : 'N U T, 0, 0, 0',
	X =	2126.823713	mm,	Y =	618.227090	mm,	Z =	688.352700	mm,
	W =	-176.966735	deg,	P =	-51.386539	deg,	R =	43.920791	deg
};
P[803]{
   GP1:
	UF : 0, UT : 1,		CONFIG : 'N U T, 0, 0, 0',
	X =	2142.478268	mm,	Y =	612.312381	mm,	Z =	698.120456	mm,
	W =	-179.425340	deg,	P =	-52.858387	deg,	R =	42.391337	deg
};
P[804]{
   GP1:
	UF : 0, UT : 1,		CONFIG : 'N U T, 0, 0, 0',
	X =	2150.343852	mm,	Y =	608.943745	mm,	Z =	703.322591	mm,
	W =	179.483862	deg,	P =	-54.171034	deg,	R =	41.446109	deg
};
P[805]{
   GP1:
	UF : 0, UT : 1,		CONFIG : 'N U T, 0, 0, 0',
	X =	2148.491543	mm,	Y =	602.062834	mm,	Z =	695.190166	mm,
	W =	149.350558	deg,	P =	-45.659355	deg,	R =	81.231272	deg
};
P[806]{
   GP1:
	UF : 0, UT : 1,		CONFIG : 'N U T, 0, 0, 0',
	X =	2132.902521	mm,	Y =	608.346374	mm,	Z =	685.238634	mm,
	W =	149.350558	deg,	P =	-45.659355	deg,	R =	81.231272	deg
};
P[807]{
   GP1:
	UF : 0, UT : 1,		CONFIG : 'N U T, 0, 0, 0',
	X =	2116.872884	mm,	Y =	613.663863	mm,	Z =	675.880479	mm,
	W =	152.007243	deg,	P =	-45.388655	deg,	R =	82.382844	deg
};
P[808]{
   GP1:
	UF : 0, UT : 1,		CONFIG : 'N U T, 0, 0, 0',
	X =	2100.249251	mm,	Y =	618.094640	mm,	Z =	667.176822	mm,
	W =	155.152979	deg,	P =	-44.232976	deg,	R =	82.958846	deg
};
P[809]{
   GP1:
	UF : 0, UT : 1,		CONFIG : 'N U T, 0, 0, 0',
	X =	2083.027426	mm,	Y =	621.356004	mm,	Z =	659.275787	mm,
	W =	158.916030	deg,	P =	-42.865821	deg,	R =	83.765156	deg
};
P[810]{
   GP1:
	UF : 0, UT : 1,		CONFIG : 'N U T, 0, 0, 0',
	X =	2065.295306	mm,	Y =	623.496703	mm,	Z =	652.095276	mm,
	W =	162.311784	deg,	P =	-42.326352	deg,	R =	84.896310	deg
};
P[811]{
   GP1:
	UF : 0, UT : 1,		CONFIG : 'N U T, 0, 0, 0',
	X =	2047.148904	mm,	Y =	624.282242	mm,	Z =	645.902844	mm,
	W =	166.497123	deg,	P =	-41.872658	deg,	R =	86.260127	deg
};
P[812]{
   GP1:
	UF : 0, UT : 1,		CONFIG : 'N U T, 0, 0, 0',
	X =	2028.682385	mm,	Y =	623.738183	mm,	Z =	640.786472	mm,
	W =	170.791821	deg,	P =	-40.898448	deg,	R =	87.435476	deg
};
P[813]{
   GP1:
	UF : 0, UT : 1,		CONFIG : 'N U T, 0, 0, 0',
	X =	2010.032713	mm,	Y =	621.847775	mm,	Z =	636.707170	mm,
	W =	175.047595	deg,	P =	-40.434450	deg,	R =	88.658437	deg
};
P[814]{
   GP1:
	UF : 0, UT : 1,		CONFIG : 'N U T, 0, 0, 0',
	X =	1991.396659	mm,	Y =	618.527935	mm,	Z =	633.831295	mm,
	W =	179.761013	deg,	P =	-39.941636	deg,	R =	89.930176	deg
};
P[815]{
   GP1:
	UF : 0, UT : 1,		CONFIG : 'N U T, 0, 0, 0',
	X =	1972.949641	mm,	Y =	613.727298	mm,	Z =	632.236088	mm,
	W =	-175.158016	deg,	P =	-39.665069	deg,	R =	91.185569	deg
};
P[816]{
   GP1:
	UF : 0, UT : 1,		CONFIG : 'N U T, 0, 0, 0',
	X =	1954.735217	mm,	Y =	607.705950	mm,	Z =	631.724723	mm,
	W =	-170.712286	deg,	P =	-39.756212	deg,	R =	92.099256	deg
};
P[817]{
   GP1:
	UF : 0, UT : 1,		CONFIG : 'N U T, 0, 0, 0',
	X =	1937.006937	mm,	Y =	600.447188	mm,	Z =	632.399858	mm,
	W =	-165.865240	deg,	P =	-39.789781	deg,	R =	92.963903	deg
};
P[818]{
   GP1:
	UF : 0, UT : 1,		CONFIG : 'N U T, 0, 0, 0',
	X =	1919.772756	mm,	Y =	592.147290	mm,	Z =	634.151754	mm,
	W =	-161.693780	deg,	P =	-39.414425	deg,	R =	93.803930	deg
};
P[819]{
   GP1:
	UF : 0, UT : 1,		CONFIG : 'N U T, 0, 0, 0',
	X =	1903.087741	mm,	Y =	582.919944	mm,	Z =	636.792237	mm,
	W =	-157.662805	deg,	P =	-39.702133	deg,	R =	94.209673	deg
};
P[820]{
   GP1:
	UF : 0, UT : 1,		CONFIG : 'N U T, 0, 0, 0',
	X =	1887.025615	mm,	Y =	572.895757	mm,	Z =	640.319984	mm,
	W =	-153.866751	deg,	P =	-39.706500	deg,	R =	94.652492	deg
};
P[821]{
   GP1:
	UF : 0, UT : 1,		CONFIG : 'N U T, 0, 0, 0',
	X =	1871.571237	mm,	Y =	562.182687	mm,	Z =	644.622034	mm,
	W =	-150.481051	deg,	P =	-39.656196	deg,	R =	95.030379	deg
};
P[822]{
   GP1:
	UF : 0, UT : 1,		CONFIG : 'N U T, 0, 0, 0',
	X =	1856.734822	mm,	Y =	550.880380	mm,	Z =	649.621791	mm,
	W =	-147.441634	deg,	P =	-39.497027	deg,	R =	95.430627	deg
};
P[823]{
   GP1:
	UF : 0, UT : 1,		CONFIG : 'N U T, 0, 0, 0',
	X =	1849.571091	mm,	Y =	545.067612	mm,	Z =	652.336911	mm,
	W =	-145.477606	deg,	P =	-39.301431	deg,	R =	95.768504	deg
};
P[824]{
   GP1:
	UF : 0, UT : 1,		CONFIG : 'N U T, 0, 0, 0',
	X =	1851.615366	mm,	Y =	538.259624	mm,	Z =	645.367223	mm,
	W =	-135.050236	deg,	P =	-21.894477	deg,	R =	72.579983	deg
};
P[825]{
   GP1:
	UF : 0, UT : 1,		CONFIG : 'N U T, 0, 0, 0',
	X =	1866.649556	mm,	Y =	549.993049	mm,	Z =	640.021729	mm,
	W =	-135.050236	deg,	P =	-21.894477	deg,	R =	72.579983	deg
};
P[826]{
   GP1:
	UF : 0, UT : 1,		CONFIG : 'N U T, 0, 0, 0',
	X =	1882.093847	mm,	Y =	561.133840	mm,	Z =	635.349619	mm,
	W =	-137.128961	deg,	P =	-22.718556	deg,	R =	71.422050	deg
};
P[827]{
   GP1:
	UF : 0, UT : 1,		CONFIG : 'N U T, 0, 0, 0',
	X =	1898.147436	mm,	Y =	571.607347	mm,	Z =	631.443364	mm,
	W =	-139.771320	deg,	P =	-23.696914	deg,	R =	70.058982	deg
};
P[828]{
   GP1:
	UF : 0, UT : 1,		CONFIG : 'N U T, 0, 0, 0',
	X =	1914.858129	mm,	Y =	581.239690	mm,	Z =	628.420088	mm,
	W =	-142.527461	deg,	P =	-25.091215	deg,	R =	68.280078	deg
};
P[829]{
   GP1:
	UF : 0, UT : 1,		CONFIG : 'N U T, 0, 0, 0',
	X =	1932.194413	mm,	Y =	589.913442	mm,	Z =	626.479948	mm,
	W =	-146.398831	deg,	P =	-26.179416	deg,	R =	66.694902	deg
};
P[830]{
   GP1:
	UF : 0, UT : 1,		CONFIG : 'N U T, 0, 0, 0',
	X =	1949.950701	mm,	Y =	598.010177	mm,	Z =	625.633210	mm,
	W =	-154.076280	deg,	P =	-23.352594	deg,	R =	67.545779	deg
};
P[831]{
   GP1:
	UF : 0, UT : 1,		CONFIG : 'N U T, 0, 0, 0',
	X =	1968.332496	mm,	Y =	604.257525	mm,	Z =	625.718061	mm,
	W =	-155.540969	deg,	P =	-27.382750	deg,	R =	63.851472	deg
};
P[832]{
   GP1:
	UF : 0, UT : 1,		CONFIG : 'N U T, 0, 0, 0',
	X =	1987.070940	mm,	Y =	609.386831	mm,	Z =	626.921606	mm,
	W =	-157.090260	deg,	P =	-30.577690	deg,	R =	61.034657	deg
};
P[833]{
   GP1:
	UF : 0, UT : 1,		CONFIG : 'N U T, 0, 0, 0',
	X =	2005.974042	mm,	Y =	613.279397	mm,	Z =	629.338698	mm,
	W =	-159.858146	deg,	P =	-33.067836	deg,	R =	58.617207	deg
};
P[834]{
   GP1:
	UF : 0, UT : 1,		CONFIG : 'N U T, 0, 0, 0',
	X =	2024.815053	mm,	Y =	615.510834	mm,	Z =	633.189270	mm,
	W =	-163.698856	deg,	P =	-35.885590	deg,	R =	55.825554	deg
};
P[835]{
   GP1:
	UF : 0, UT : 1,		CONFIG : 'N U T, 0, 0, 0',
	X =	2043.581866	mm,	Y =	616.369806	mm,	Z =	638.165099	mm,
	W =	-166.819138	deg,	P =	-38.185996	deg,	R =	53.599760	deg
};
P[836]{
   GP1:
	UF : 0, UT : 1,		CONFIG : 'N U T, 0, 0, 0',
	X =	2062.065141	mm,	Y =	615.834319	mm,	Z =	644.199867	mm,
	W =	-169.614560	deg,	P =	-40.750324	deg,	R =	51.350208	deg
};
P[837]{
   GP1:
	UF : 0, UT : 1,		CONFIG : 'N U T, 0, 0, 0',
	X =	2080.090857	mm,	Y =	613.932309	mm,	Z =	651.252496	mm,
	W =	-172.396436	deg,	P =	-43.311562	deg,	R =	49.143827	deg
};
P[838]{
   GP1:
	UF : 0, UT : 1,		CONFIG : 'N U T, 0, 0, 0',
	X =	2097.577842	mm,	Y =	610.772764	mm,	Z =	659.217570	mm,
	W =	-175.093846	deg,	P =	-45.578693	deg,	R =	47.117239	deg
};
P[839]{
   GP1:
	UF : 0, UT : 1,		CONFIG : 'N U T, 0, 0, 0',
	X =	2114.574090	mm,	Y =	606.538730	mm,	Z =	667.867887	mm,
	W =	-176.810481	deg,	P =	-47.964198	deg,	R =	45.406767	deg
};
P[840]{
   GP1:
	UF : 0, UT : 1,		CONFIG : 'N U T, 0, 0, 0',
	X =	2130.850172	mm,	Y =	601.227981	mm,	Z =	677.231203	mm,
	W =	-178.837703	deg,	P =	-50.396925	deg,	R =	43.579965	deg
};
P[841]{
   GP1:
	UF : 0, UT : 1,		CONFIG : 'N U T, 0, 0, 0',
	X =	2146.590253	mm,	Y =	595.118781	mm,	Z =	687.145470	mm,
	W =	179.337405	deg,	P =	-51.856761	deg,	R =	42.203446	deg
};
P[842]{
   GP1:
	UF : 0, UT : 1,		CONFIG : 'N U T, 0, 0, 0',
	X =	2144.657267	mm,	Y =	588.010945	mm,	Z =	679.172536	mm,
	W =	150.474945	deg,	P =	-44.167395	deg,	R =	80.403319	deg
};
P[843]{
   GP1:
	UF : 0, UT : 1,		CONFIG : 'N U T, 0, 0, 0',
	X =	2128.576754	mm,	Y =	594.194085	mm,	Z =	669.157912	mm,
	W =	150.474945	deg,	P =	-44.167395	deg,	R =	80.403319	deg
};
P[844]{
   GP1:
	UF : 0, UT : 1,		CONFIG : 'N U T, 0, 0, 0',
	X =	2111.990480	mm,	Y =	599.228955	mm,	Z =	659.905093	mm,
	W =	153.680707	deg,	P =	-43.339689	deg,	R =	81.530719	deg
};
P[845]{
   GP1:
	UF : 0, UT : 1,		CONFIG : 'N U T, 0, 0, 0',
	X =	2094.815677	mm,	Y =	603.405894	mm,	Z =	651.233012	mm,
	W =	156.468910	deg,	P =	-42.395069	deg,	R =	82.317026	deg
};
P[846]{
   GP1:
	UF : 0, UT : 1,		CONFIG : 'N U T, 0, 0, 0',
	X =	2077.078381	mm,	Y =	606.283673	mm,	Z =	643.406603	mm,
	W =	160.174460	deg,	P =	-41.891132	deg,	R =	83.790014	deg
};
P[847]{
   GP1:
	UF : 0, UT : 1,		CONFIG : 'N U T, 0, 0, 0',
	X =	2058.815719	mm,	Y =	608.005957	mm,	Z =	636.458501	mm,
	W =	163.811579	deg,	P =	-40.855594	deg,	R =	84.887446	deg
};
P[848]{
   GP1:
	UF : 0, UT : 1,		CONFIG : 'N U T, 0, 0, 0',
	X =	2040.159846	mm,	Y =	608.280329	mm,	Z =	630.582754	mm,
	W =	168.107760	deg,	P =	-39.930311	deg,	R =	86.292997	deg
};
P[849]{
   GP1:
	UF : 0, UT : 1,		CONFIG : 'N U T, 0, 0, 0',
	X =	2021.135138	mm,	Y =	607.506202	mm,	Z =	626.226826	mm,
	W =	171.616624	deg,	P =	-30.899337	deg,	R =	86.443968	deg
};
P[850]{
   GP1:
	UF : 0, UT : 1,		CONFIG : 'N U T, 0, 0, 0',
	X =	2001.988310	mm,	Y =	605.181579	mm,	Z =	622.948826	mm,
	W =	174.477127	deg,	P =	-23.689275	deg,	R =	88.036999	deg
};
P[851]{
   GP1:
	UF : 0, UT : 1,		CONFIG : 'N U T, 0, 0, 0',
	X =	1983.308899	mm,	Y =	600.024510	mm,	Z =	620.415761	mm,
	W =	-177.923887	deg,	P =	-36.275132	deg,	R =	90.944175	deg
};
P[852]{
   GP1:
	UF : 0, UT : 1,		CONFIG : 'N U T, 0, 0, 0',
	X =	1964.850233	mm,	Y =	593.949197	mm,	Z =	619.998813	mm,
	W =	-172.373674	deg,	P =	-34.652376	deg,	R =	93.082846	deg
};
P[853]{
   GP1:
	UF : 0, UT : 1,		CONFIG : 'N U T, 0, 0, 0',
	X =	1946.190064	mm,	Y =	587.448123	mm,	Z =	620.298093	mm,
	W =	-172.006402	deg,	P =	-29.550035	deg,	R =	94.686048	deg
};
P[854]{
   GP1:
	UF : 0, UT : 1,		CONFIG : 'N U T, 0, 0, 0',
	X =	1927.905948	mm,	Y =	580.024088	mm,	Z =	620.982468	mm,
	W =	-169.842455	deg,	P =	-29.844058	deg,	R =	95.536298	deg
};
P[855]{
   GP1:
	UF : 0, UT : 1,		CONFIG : 'N U T, 0, 0, 0',
	X =	1910.721826	mm,	Y =	571.242756	mm,	Z =	623.387676	mm,
	W =	-165.229640	deg,	P =	-26.846936	deg,	R =	98.881301	deg
};
P[856]{
   GP1:
	UF : 0, UT : 1,		CONFIG : 'N U T, 0, 0, 0',
	X =	1893.738949	mm,	Y =	560.296793	mm,	Z =	626.314042	mm,
	W =	-156.222105	deg,	P =	-38.074436	deg,	R =	95.448819	deg
};
P[857]{
   GP1:
	UF : 0, UT : 1,		CONFIG : 'N U T, 0, 0, 0',
	X =	1884.250248	mm,	Y =	554.073906	mm,	Z =	628.550842	mm,
	W =	-153.101874	deg,	P =	-38.984533	deg,	R =	95.263261	deg
};
P[858]{
   GP1:
	UF : 0, UT : 1,		CONFIG : 'N U T, 0, 0, 0',
	X =	1866.111827	mm,	Y =	540.973975	mm,	Z =	634.031217	mm,
	W =	-149.536564	deg,	P =	-39.137116	deg,	R =	95.547881	deg
};
P[859]{
   GP1:
	UF : 0, UT : 1,		CONFIG : 'N U T, 0, 0, 0',
	X =	1858.614647	mm,	Y =	535.196992	mm,	Z =	636.612256	mm,
	W =	-147.484335	deg,	P =	-38.969883	deg,	R =	95.899116	deg
};
P[860]{
   GP1:
	UF : 0, UT : 1,		CONFIG : 'N U T, 0, 0, 0',
	X =	1936.561677	mm,	Y =	571.380063	mm,	Z =	617.369556	mm,
	W =	-172.389357	deg,	P =	-31.226715	deg,	R =	94.029203	deg
};
P[861]{
   GP1:
	UF : 0, UT : 1,		CONFIG : 'N U T, 0, 0, 0',
	X =	1947.980778	mm,	Y =	575.349462	mm,	Z =	617.460185	mm,
	W =	-172.389357	deg,	P =	-31.226715	deg,	R =	94.029203	deg
};
P[862]{
   GP1:
	UF : 0, UT : 1,		CONFIG : 'N U T, 0, 0, 0',
	X =	1967.450400	mm,	Y =	581.537827	mm,	Z =	617.161212	mm,
	W =	168.569288	deg,	P =	-41.016388	deg,	R =	125.777102	deg
};
P[863]{
   GP1:
	UF : 0, UT : 1,		CONFIG : 'N U T, 0, 0, 0',
	X =	1985.948855	mm,	Y =	587.960340	mm,	Z =	617.314605	mm,
	W =	168.569288	deg,	P =	-41.016388	deg,	R =	125.777102	deg
};
P[864]{
   GP1:
	UF : 0, UT : 1,		CONFIG : 'N U T, 0, 0, 0',
	X =	2003.617365	mm,	Y =	594.519557	mm,	Z =	618.351050	mm,
	W =	171.833346	deg,	P =	-27.562577	deg,	R =	122.555661	deg
};
P[865]{
   GP1:
	UF : 0, UT : 1,		CONFIG : 'N U T, 0, 0, 0',
	X =	2022.069587	mm,	Y =	598.400911	mm,	Z =	620.250948	mm,
	W =	165.229046	deg,	P =	-30.603979	deg,	R =	120.770963	deg
};
P[866]{
   GP1:
	UF : 0, UT : 1,		CONFIG : 'N U T, 0, 0, 0',
	X =	2040.233328	mm,	Y =	600.878137	mm,	Z =	624.678533	mm,
	W =	162.522222	deg,	P =	-18.327737	deg,	R =	112.953907	deg
};
P[867]{
   GP1:
	UF : 0, UT : 1,		CONFIG : 'N U T, 0, 0, 0',
	X =	2058.570721	mm,	Y =	599.873871	mm,	Z =	629.883448	mm,
	W =	151.913285	deg,	P =	-29.754802	deg,	R =	114.901783	deg
};
P[868]{
   GP1:
	UF : 0, UT : 1,		CONFIG : 'N U T, 0, 0, 0',
	X =	2076.448996	mm,	Y =	598.289347	mm,	Z =	636.629065	mm,
	W =	148.068773	deg,	P =	-28.993299	deg,	R =	112.543235	deg
};
P[869]{
   GP1:
	UF : 0, UT : 1,		CONFIG : 'N U T, 0, 0, 0',
	X =	2093.846385	mm,	Y =	595.451715	mm,	Z =	644.264593	mm,
	W =	144.620247	deg,	P =	-28.567946	deg,	R =	110.466184	deg
};
P[870]{
   GP1:
	UF : 0, UT : 1,		CONFIG : 'N U T, 0, 0, 0',
	X =	2110.712146	mm,	Y =	591.533411	mm,	Z =	652.669951	mm,
	W =	141.719237	deg,	P =	-28.080435	deg,	R =	108.381744	deg
};
P[871]{
   GP1:
	UF : 0, UT : 1,		CONFIG : 'N U T, 0, 0, 0',
	X =	2127.009975	mm,	Y =	586.602805	mm,	Z =	661.711654	mm,
	W =	138.853144	deg,	P =	-28.059736	deg,	R =	106.739673	deg
};
P[872]{
   GP1:
	UF : 0, UT : 1,		CONFIG : 'N U T, 0, 0, 0',
	X =	2142.704026	mm,	Y =	580.764992	mm,	Z =	671.302791	mm,
	W =	136.022512	deg,	P =	-28.349160	deg,	R =	105.478700	deg
};
P[873]{
   GP1:
	UF : 0, UT : 1,		CONFIG : 'N U T, 0, 0, 0',
	X =	2140.432209	mm,	Y =	573.487960	mm,	Z =	663.413620	mm,
	W =	130.724090	deg,	P =	-8.547436	deg,	R =	123.967225	deg
};
P[874]{
   GP1:
	UF : 0, UT : 1,		CONFIG : 'N U T, 0, 0, 0',
	X =	2124.597057	mm,	Y =	579.256056	mm,	Z =	653.821116	mm,
	W =	130.724090	deg,	P =	-8.547436	deg,	R =	123.967225	deg
};
P[875]{
   GP1:
	UF : 0, UT : 1,		CONFIG : 'N U T, 0, 0, 0',
	X =	2108.323828	mm,	Y =	583.972710	mm,	Z =	644.934892	mm,
	W =	132.861387	deg,	P =	-9.507073	deg,	R =	126.751853	deg
};
P[876]{
   GP1:
	UF : 0, UT : 1,		CONFIG : 'N U T, 0, 0, 0',
	X =	2091.475429	mm,	Y =	587.722980	mm,	Z =	636.696020	mm,
	W =	135.058774	deg,	P =	-10.552104	deg,	R =	129.460171	deg
};
P[877]{
   GP1:
	UF : 0, UT : 1,		CONFIG : 'N U T, 0, 0, 0',
	X =	2074.101287	mm,	Y =	590.353887	mm,	Z =	629.235571	mm,
	W =	137.488986	deg,	P =	-11.868364	deg,	R =	132.439309	deg
};
P[878]{
   GP1:
	UF : 0, UT : 1,		CONFIG : 'N U T, 0, 0, 0',
	X =	2056.116313	mm,	Y =	592.693766	mm,	Z =	623.336009	mm,
	W =	152.533882	deg,	P =	-2.096782	deg,	R =	128.263831	deg
};
P[879]{
   GP1:
	UF : 0, UT : 1,		CONFIG : 'N U T, 0, 0, 0',
	X =	2038.137540	mm,	Y =	589.764435	mm,	Z =	619.163308	mm,
	W =	150.183475	deg,	P =	-15.892358	deg,	R =	142.138420	deg
};
P[880]{
   GP1:
	UF : 0, UT : 1,		CONFIG : 'N U T, 0, 0, 0',
	X =	2021.746962	mm,	Y =	586.474182	mm,	Z =	618.080853	mm,
	W =	164.762805	deg,	P =	-10.567016	deg,	R =	144.584221	deg
};
P[881]{
   GP1:
	UF : 0, UT : 1,		CONFIG : 'N U T, 0, 0, 0',
	X =	2003.425408	mm,	Y =	581.329739	mm,	Z =	618.063313	mm,
	W =	178.460626	deg,	P =	-0.886054	deg,	R =	147.370644	deg
};
P[882]{
   GP1:
	UF : 0, UT : 1,		CONFIG : 'N U T, 0, 0, 0',
	X =	1985.013396	mm,	Y =	574.969738	mm,	Z =	617.881286	mm,
	W =	178.535374	deg,	P =	-0.984171	deg,	R =	147.503956	deg
};
P[883]{
   GP1:
	UF : 0, UT : 1,		CONFIG : 'N U T, 0, 0, 0',
	X =	1975.935528	mm,	Y =	571.838370	mm,	Z =	617.790300	mm,
	W =	178.543393	deg,	P =	-0.961790	deg,	R =	147.494977	deg
};
P[884]{
   GP1:
	UF : 0, UT : 1,		CONFIG : 'N U T, 0, 0, 0',
	X =	2015.231747	mm,	Y =	569.989378	mm,	Z =	617.728739	mm,
	W =	178.193057	deg,	P =	-0.073673	deg,	R =	172.574110	deg
};
P[885]{
   GP1:
	UF : 0, UT : 1,		CONFIG : 'N U T, 0, 0, 0',
	X =	2024.281449	mm,	Y =	573.074938	mm,	Z =	617.851137	mm,
	W =	178.193057	deg,	P =	-0.073673	deg,	R =	172.574110	deg
};
P[886]{
   GP1:
	UF : 0, UT : 1,		CONFIG : 'N U T, 0, 0, 0',
	X =	2041.762600	mm,	Y =	578.977173	mm,	Z =	618.085021	mm,
	W =	177.481010	deg,	P =	-0.425930	deg,	R =	172.588775	deg
};
P[887]{
   GP1:
	UF : 0, UT : 1,		CONFIG : 'N U T, 0, 0, 0',
	X =	2058.412081	mm,	Y =	581.890099	mm,	Z =	619.230036	mm,
	W =	158.657744	deg,	P =	-4.944196	deg,	R =	169.848488	deg
};
P[888]{
   GP1:
	UF : 0, UT : 1,		CONFIG : 'N U T, 0, 0, 0',
	X =	2075.345606	mm,	Y =	582.440266	mm,	Z =	623.756835	mm,
	W =	151.783764	deg,	P =	2.965468	deg,	R =	158.638329	deg
};
P[889]{
   GP1:
	UF : 0, UT : 1,		CONFIG : 'N U T, 0, 0, 0',
	X =	2091.670644	mm,	Y =	579.406024	mm,	Z =	630.405831	mm,
	W =	137.650948	deg,	P =	5.780487	deg,	R =	150.808271	deg
};
P[890]{
   GP1:
	UF : 0, UT : 1,		CONFIG : 'N U T, 0, 0, 0',
	X =	2107.857485	mm,	Y =	575.818823	mm,	Z =	638.314606	mm,
	W =	135.664769	deg,	P =	7.873459	deg,	R =	146.936630	deg
};
P[891]{
   GP1:
	UF : 0, UT : 1,		CONFIG : 'N U T, 0, 0, 0',
	X =	2123.581638	mm,	Y =	571.317155	mm,	Z =	646.821987	mm,
	W =	133.765412	deg,	P =	9.345894	deg,	R =	143.845165	deg
};
P[892]{
   GP1:
	UF : 0, UT : 1,		CONFIG : 'N U T, 0, 0, 0',
	X =	2138.671167	mm,	Y =	565.943371	mm,	Z =	655.928473	mm,
	W =	132.202477	deg,	P =	10.961554	deg,	R =	140.309444	deg
};
P[893]{
   GP1:
	UF : 0, UT : 1,		CONFIG : 'N U T, 0, 0, 0',
	X =	2138.551566	mm,	Y =	557.587191	mm,	Z =	649.508320	mm,
	W =	131.817631	deg,	P =	-8.026197	deg,	R =	123.569090	deg
};
P[894]{
   GP1:
	UF : 0, UT : 1,		CONFIG : 'N U T, 0, 0, 0',
	X =	2122.899934	mm,	Y =	563.156300	mm,	Z =	640.137993	mm,
	W =	131.817631	deg,	P =	-8.026197	deg,	R =	123.569090	deg
};
P[895]{
   GP1:
	UF : 0, UT : 1,		CONFIG : 'N U T, 0, 0, 0',
	X =	2106.826722	mm,	Y =	567.690106	mm,	Z =	631.476626	mm,
	W =	134.061047	deg,	P =	-8.910523	deg,	R =	126.312662	deg
};
P[896]{
   GP1:
	UF : 0, UT : 1,		CONFIG : 'N U T, 0, 0, 0',
	X =	2090.142464	mm,	Y =	571.853323	mm,	Z =	623.849423	mm,
	W =	143.595196	deg,	P =	-3.654324	deg,	R =	123.821052	deg
};
P[897]{
   GP1:
	UF : 0, UT : 1,		CONFIG : 'N U T, 0, 0, 0',
	X =	2072.846348	mm,	Y =	571.852603	mm,	Z =	618.562659	mm,
	W =	151.264771	deg,	P =	-7.374624	deg,	R =	133.561325	deg
};
P[898]{
   GP1:
	UF : 0, UT : 1,		CONFIG : 'N U T, 0, 0, 0',
	X =	2057.123273	mm,	Y =	568.873859	mm,	Z =	617.816601	mm,
	W =	175.471624	deg,	P =	1.028997	deg,	R =	143.408241	deg
};
P[899]{
   GP1:
	UF : 0, UT : 1,		CONFIG : 'N U T, 0, 0, 0',
	X =	2039.279991	mm,	Y =	562.808020	mm,	Z =	617.573630	mm,
	W =	178.386233	deg,	P =	-0.806491	deg,	R =	147.250783	deg
};
P[900]{
   GP1:
	UF : 0, UT : 1,		CONFIG : 'N U T, 0, 0, 0',
	X =	2085.846492	mm,	Y =	561.436044	mm,	Z =	617.480241	mm,
	W =	146.304700	deg,	P =	4.668136	deg,	R =	154.734213	deg
};
P[901]{
   GP1:
	UF : 0, UT : 1,		CONFIG : 'N U T, 0, 0, 0',
	X =	2093.522748	mm,	Y =	561.111940	mm,	Z =	620.054237	mm,
	W =	146.304700	deg,	P =	4.668136	deg,	R =	154.734213	deg
};
P[902]{
   GP1:
	UF : 0, UT : 1,		CONFIG : 'N U T, 0, 0, 0',
	X =	2108.694093	mm,	Y =	558.849494	mm,	Z =	626.302552	mm,
	W =	141.130259	deg,	P =	6.757329	deg,	R =	150.218047	deg
};
P[903]{
   GP1:
	UF : 0, UT : 1,		CONFIG : 'N U T, 0, 0, 0',
	X =	2122.858212	mm,	Y =	554.702256	mm,	Z =	633.894408	mm,
	W =	135.110311	deg,	P =	9.755662	deg,	R =	143.487460	deg
};
P[904]{
   GP1:
	UF : 0, UT : 1,		CONFIG : 'N U T, 0, 0, 0',
	X =	2136.729929	mm,	Y =	549.756750	mm,	Z =	642.210257	mm,
	W =	132.906395	deg,	P =	11.147195	deg,	R =	140.162629	deg
};
P[905]{
   GP1:
	UF : 0, UT : 1,		CONFIG : 'N U T, 0, 0, 0',
	X =	2124.410034	mm,	Y =	545.521303	mm,	Z =	628.717145	mm,
	W =	133.381973	deg,	P =	11.251611	deg,	R =	140.110422	deg
};
P[906]{
   GP1:
	UF : 0, UT : 1,		CONFIG : 'N U T, 0, 0, 0',
	X =	2132.997690	mm,	Y =	542.484044	mm,	Z =	633.842996	mm,
	W =	133.381973	deg,	P =	11.251611	deg,	R =	140.110422	deg
};
P[907]{
   GP1:
	UF : 0, UT : 1,		CONFIG : 'N U T, 0, 0, 0',
	X =	2121.706023	mm,	Y =	546.392903	mm,	Z =	627.161754	mm,
	W =	140.649912	deg,	P =	29.185130	deg,	R =	160.868312	deg
};
P[908]{
   GP1:
	UF : 0, UT : 1,		CONFIG : 'N U T, 0, 0, 0',
	X =	2106.005631	mm,	Y =	550.422884	mm,	Z =	620.133194	mm,
	W =	156.646090	deg,	P =	24.944585	deg,	R =	168.210205	deg
};
P[909]{
   GP1:
	UF : 0, UT : 1,		CONFIG : 'N U T, 0, 0, 0',
	X =	2094.505214	mm,	Y =	542.699496	mm,	Z =	640.944003	mm,
	W =	156.646090	deg,	P =	24.944585	deg,	R =	168.210205	deg
};

/END.
